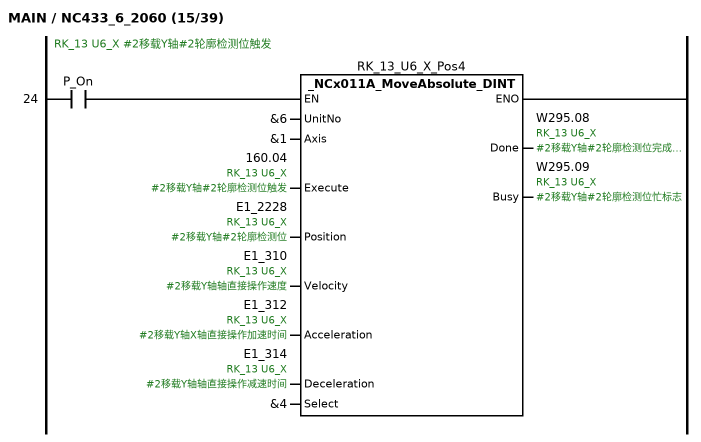
; [picture p240: MAIN / NC433_6_2060, rungs 24-24]
; rung 24: RK_13 U6_X #2移载Y轴#2轮廓检测位触发
LD P_On
CALL RK_13_U6_X_Pos4 : _NCx011A_MoveAbsolute_DINT (UnitNo := &6, Axis := &1, Execute := 160.04, Position := E1_2228, Velocity := E1_310, Acceleration := E1_312, Deceleration := E1_314, Select := &4, Done => W295.08, Busy => W295.09)  ; RK_13 U6_X #2移载Y轴#2轮廓检测位触发, RK_13 U6_X #2移载Y轴#2轮廓检测位, RK_13 U6_X #2移载Y轴轴直接操作速度, RK_13 U6_X #2移载Y轴X轴直接操作加速时间, RK_13 U6_X #2移载Y轴轴直接操作减速时间, RK_13 U6_X #2移载Y轴#2轮廓检测位完成标志, RK_13 U6_X #2移载Y轴#2轮廓检测位忙标志

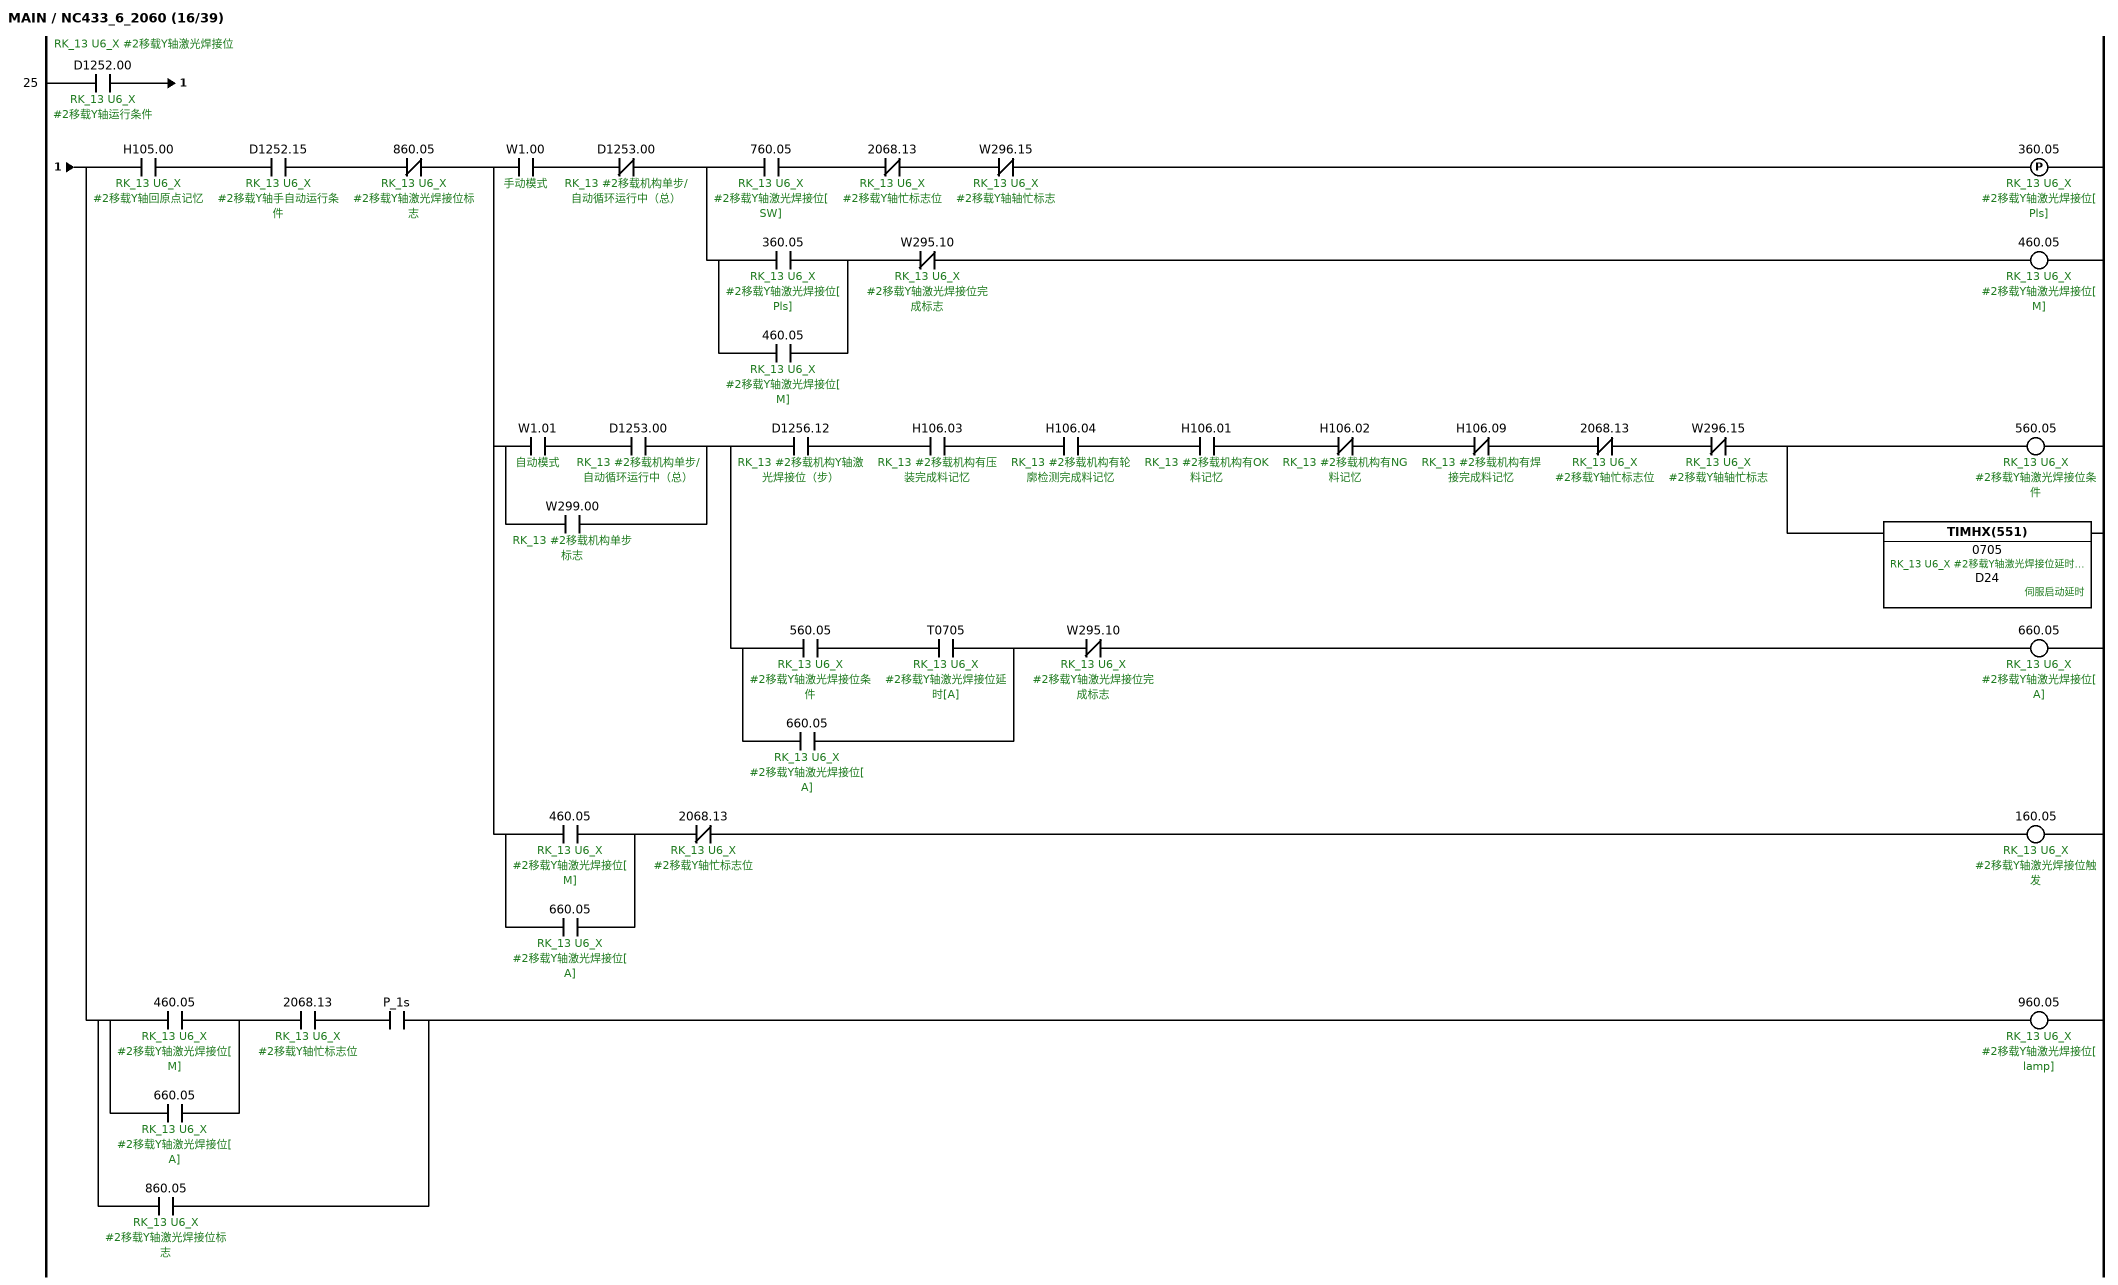
; rung 25: RK_13 U6_X #2移载Y轴激光焊接位
LD D1252.00  ; RK_13 U6_X #2移载Y轴运行条件
OUT TR0
AND H105.00  ; RK_13 U6_X #2移载Y轴回原点记忆
AND D1252.15  ; RK_13 U6_X #2移载Y轴手自动运行条件
ANDNOT 860.05  ; RK_13 U6_X #2移载Y轴激光焊接位标志
OUT TR1
AND W1.00  ; 手动模式
ANDNOT D1253.00  ; RK_13 #2移载机构单步/自动循环运行中（总）
OUT TR2
AND 760.05  ; RK_13 U6_X #2移载Y轴激光焊接位[SW]
ANDNOT 2068.13  ; RK_13 U6_X #2移载Y轴忙标志位
ANDNOT W296.15  ; RK_13 U6_X #2移载Y轴轴忙标志
DIFU(013) 360.05  ; RK_13 U6_X #2移载Y轴激光焊接位[Pls]
LD TR2
LD 360.05  ; RK_13 U6_X #2移载Y轴激光焊接位[Pls]
OR 460.05  ; RK_13 U6_X #2移载Y轴激光焊接位[M]
ANDLD
ANDNOT W295.10  ; RK_13 U6_X #2移载Y轴激光焊接位完成标志
OUT 460.05  ; RK_13 U6_X #2移载Y轴激光焊接位[M]
LD TR1
LD W1.01  ; 自动模式
AND D1253.00  ; RK_13 #2移载机构单步/自动循环运行中（总）
OR W299.00  ; RK_13 #2移载机构单步标志
ANDLD
OUT TR2
AND D1256.12  ; RK_13 #2移载机构Y轴激光焊接位（步）
AND H106.03  ; RK_13 #2移载机构有压装完成料记忆
AND H106.04  ; RK_13 #2移载机构有轮廓检测完成料记忆
AND H106.01  ; RK_13 #2移载机构有OK料记忆
ANDNOT H106.02  ; RK_13 #2移载机构有NG料记忆
ANDNOT H106.09  ; RK_13 #2移载机构有焊接完成料记忆
ANDNOT 2068.13  ; RK_13 U6_X #2移载Y轴忙标志位
ANDNOT W296.15  ; RK_13 U6_X #2移载Y轴轴忙标志
OUT 560.05  ; RK_13 U6_X #2移载Y轴激光焊接位条件
TIMHX(551) 0705 D24  ; 伺服启动延时, RK_13 U6_X #2移载Y轴激光焊接位延时[A]
LD TR2
LD 560.05  ; RK_13 U6_X #2移载Y轴激光焊接位条件
AND T0705  ; RK_13 U6_X #2移载Y轴激光焊接位延时[A]
OR 660.05  ; RK_13 U6_X #2移载Y轴激光焊接位[A]
ANDLD
ANDNOT W295.10  ; RK_13 U6_X #2移载Y轴激光焊接位完成标志
OUT 660.05  ; RK_13 U6_X #2移载Y轴激光焊接位[A]
LD TR1
LD 460.05  ; RK_13 U6_X #2移载Y轴激光焊接位[M]
OR 660.05  ; RK_13 U6_X #2移载Y轴激光焊接位[A]
ANDLD
ANDNOT 2068.13  ; RK_13 U6_X #2移载Y轴忙标志位
OUT 160.05  ; RK_13 U6_X #2移载Y轴激光焊接位触发
LD TR0
LD 460.05  ; RK_13 U6_X #2移载Y轴激光焊接位[M]
OR 660.05  ; RK_13 U6_X #2移载Y轴激光焊接位[A]
AND 2068.13  ; RK_13 U6_X #2移载Y轴忙标志位
AND P_1s
OR 860.05  ; RK_13 U6_X #2移载Y轴激光焊接位标志
ANDLD
OUT 960.05  ; RK_13 U6_X #2移载Y轴激光焊接位[lamp]

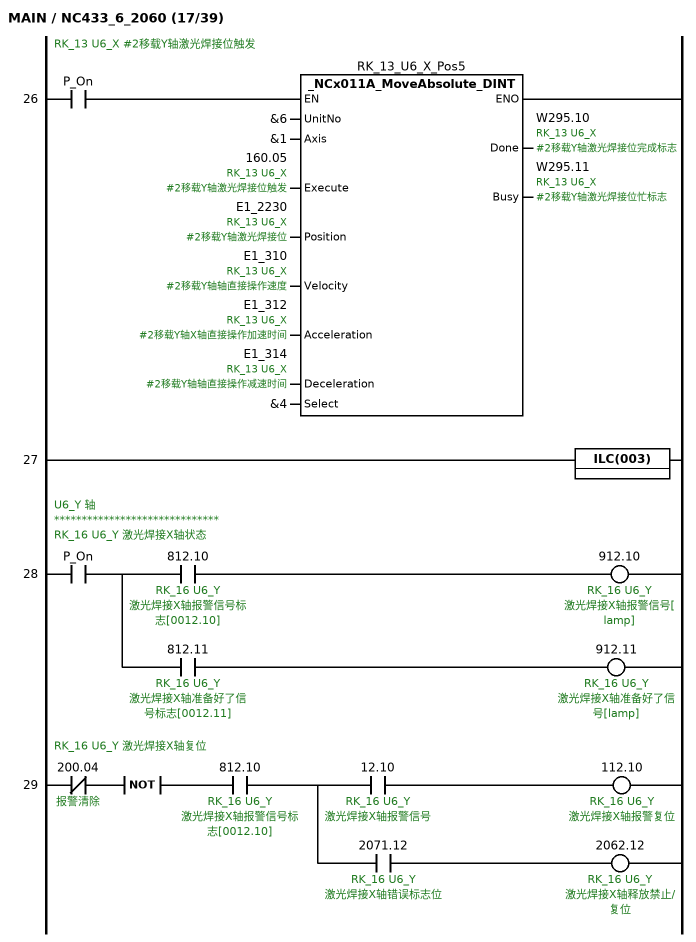
; rung 26: RK_13 U6_X #2移载Y轴激光焊接位触发
LD P_On
CALL RK_13_U6_X_Pos5 : _NCx011A_MoveAbsolute_DINT (UnitNo := &6, Axis := &1, Execute := 160.05, Position := E1_2230, Velocity := E1_310, Acceleration := E1_312, Deceleration := E1_314, Select := &4, Done => W295.10, Busy => W295.11)  ; RK_13 U6_X #2移载Y轴激光焊接位触发, RK_13 U6_X #2移载Y轴激光焊接位, RK_13 U6_X #2移载Y轴轴直接操作速度, RK_13 U6_X #2移载Y轴X轴直接操作加速时间, RK_13 U6_X #2移载Y轴轴直接操作减速时间, RK_13 U6_X #2移载Y轴激光焊接位完成标志, RK_13 U6_X #2移载Y轴激光焊接位忙标志
; rung 27
ILC(003)
; rung 28: U6_Y 轴 / ****************************** / RK_16 U6_Y 激光焊接X轴状态
LD P_On
OUT TR0
AND 812.10  ; RK_16 U6_Y 激光焊接X轴报警信号标志[0012.10]
OUT 912.10  ; RK_16 U6_Y 激光焊接X轴报警信号[lamp]
LD TR0
AND 812.11  ; RK_16 U6_Y 激光焊接X轴准备好了信号标志[0012.11]
OUT 912.11  ; RK_16 U6_Y 激光焊接X轴准备好了信号[lamp]
; rung 29: RK_16 U6_Y 激光焊接X轴复位
LDNOT 200.04  ; 报警清除
NOT(520)
AND 812.10  ; RK_16 U6_Y 激光焊接X轴报警信号标志[0012.10]
OUT TR0
AND 12.10  ; RK_16 U6_Y 激光焊接X轴报警信号
OUT 112.10  ; RK_16 U6_Y 激光焊接X轴报警复位
LD TR0
AND 2071.12  ; RK_16 U6_Y 激光焊接X轴错误标志位
OUT 2062.12  ; RK_16 U6_Y 激光焊接X轴释放禁止/复位

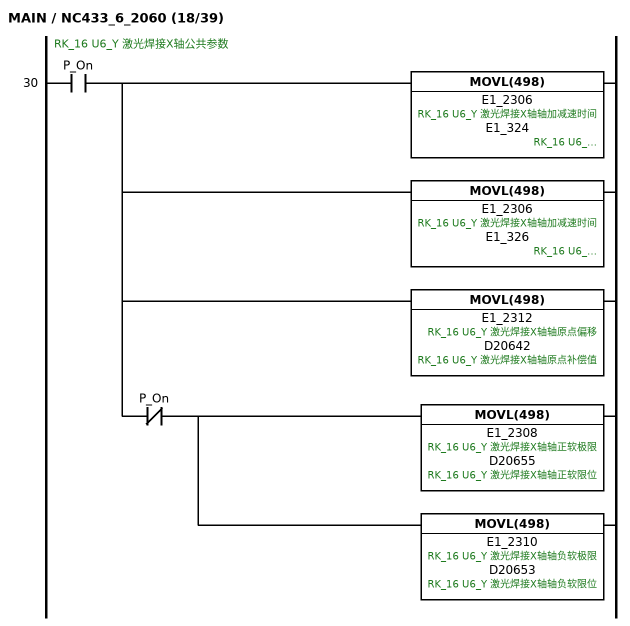
; rung 30: RK_16 U6_Y 激光焊接X轴公共参数
LD P_On
MOVL(498) E1_2306 E1_324  ; RK_16 U6_Y 激光焊接X轴轴加减速时间, RK_16 U6_Y 激光焊接X轴轴直接操作加速时间
MOVL(498) E1_2306 E1_326  ; RK_16 U6_Y 激光焊接X轴轴加减速时间, RK_16 U6_Y 激光焊接X轴轴直接操作减速时间
MOVL(498) E1_2312 D20642  ; RK_16 U6_Y 激光焊接X轴轴原点偏移, RK_16 U6_Y 激光焊接X轴轴原点补偿值
ANDNOT P_On
MOVL(498) E1_2308 D20655  ; RK_16 U6_Y 激光焊接X轴轴正软极限, RK_16 U6_Y 激光焊接X轴轴正软限位
MOVL(498) E1_2310 D20653  ; RK_16 U6_Y 激光焊接X轴轴负软极限, RK_16 U6_Y 激光焊接X轴轴负软限位

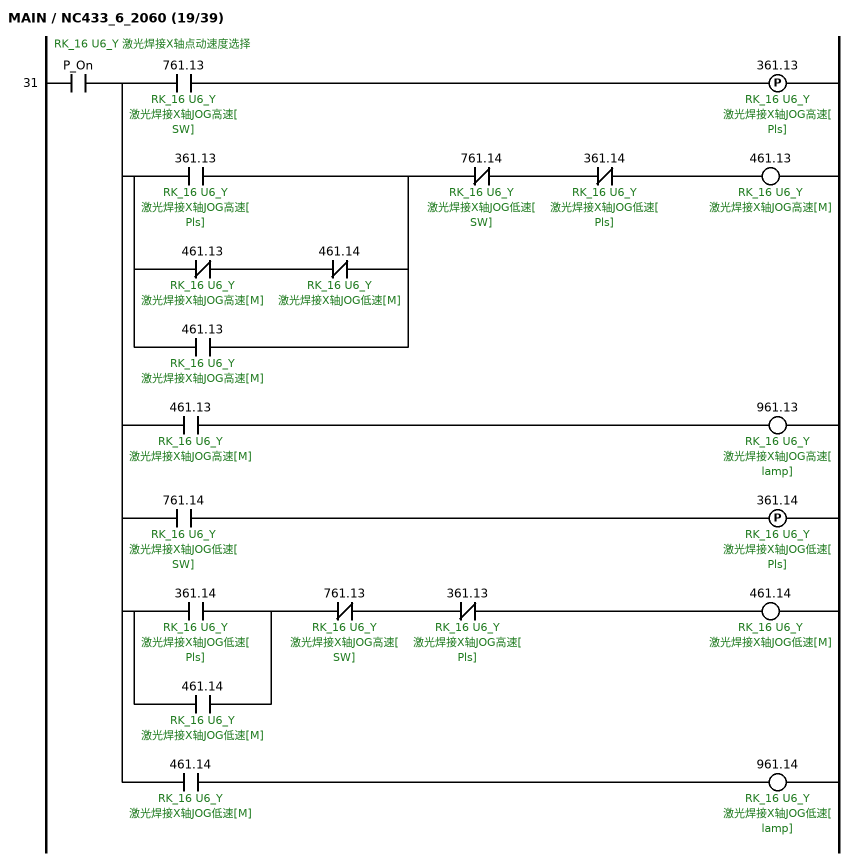
; rung 31: RK_16 U6_Y 激光焊接X轴点动速度选择
LD P_On
OUT TR0
AND 761.13  ; RK_16 U6_Y 激光焊接X轴JOG高速[SW]
DIFU(013) 361.13  ; RK_16 U6_Y 激光焊接X轴JOG高速[Pls]
LD TR0
LD 361.13  ; RK_16 U6_Y 激光焊接X轴JOG高速[Pls]
LDNOT 461.13  ; RK_16 U6_Y 激光焊接X轴JOG高速[M]
ANDNOT 461.14  ; RK_16 U6_Y 激光焊接X轴JOG低速[M]
ORLD
OR 461.13  ; RK_16 U6_Y 激光焊接X轴JOG高速[M]
ANDLD
ANDNOT 761.14  ; RK_16 U6_Y 激光焊接X轴JOG低速[SW]
ANDNOT 361.14  ; RK_16 U6_Y 激光焊接X轴JOG低速[Pls]
OUT 461.13  ; RK_16 U6_Y 激光焊接X轴JOG高速[M]
LD TR0
AND 461.13  ; RK_16 U6_Y 激光焊接X轴JOG高速[M]
OUT 961.13  ; RK_16 U6_Y 激光焊接X轴JOG高速[lamp]
LD TR0
AND 761.14  ; RK_16 U6_Y 激光焊接X轴JOG低速[SW]
DIFU(013) 361.14  ; RK_16 U6_Y 激光焊接X轴JOG低速[Pls]
LD TR0
LD 361.14  ; RK_16 U6_Y 激光焊接X轴JOG低速[Pls]
OR 461.14  ; RK_16 U6_Y 激光焊接X轴JOG低速[M]
ANDLD
ANDNOT 761.13  ; RK_16 U6_Y 激光焊接X轴JOG高速[SW]
ANDNOT 361.13  ; RK_16 U6_Y 激光焊接X轴JOG高速[Pls]
OUT 461.14  ; RK_16 U6_Y 激光焊接X轴JOG低速[M]
LD TR0
AND 461.14  ; RK_16 U6_Y 激光焊接X轴JOG低速[M]
OUT 961.14  ; RK_16 U6_Y 激光焊接X轴JOG低速[lamp]

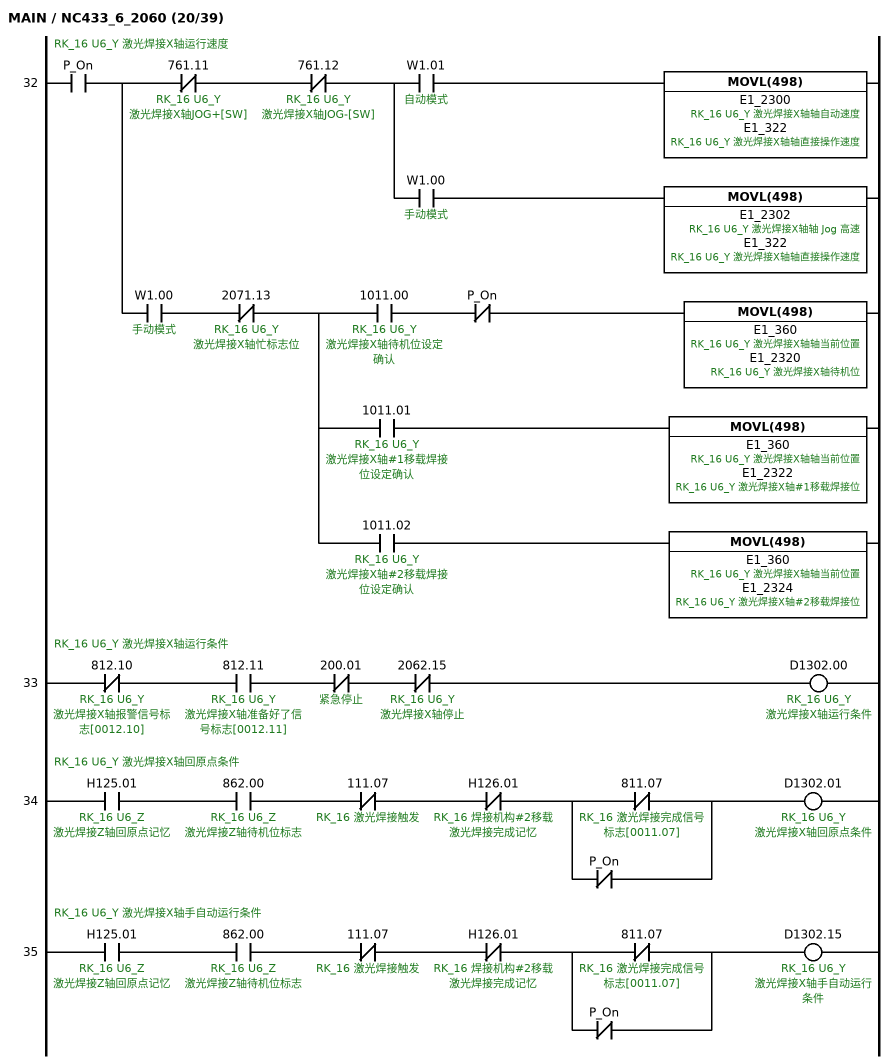
; rung 32: RK_16 U6_Y 激光焊接X轴运行速度
LD P_On
OUT TR0
ANDNOT 761.11  ; RK_16 U6_Y 激光焊接X轴JOG+[SW]
ANDNOT 761.12  ; RK_16 U6_Y 激光焊接X轴JOG-[SW]
OUT TR1
AND W1.01  ; 自动模式
MOVL(498) E1_2300 E1_322  ; RK_16 U6_Y 激光焊接X轴轴自动速度, RK_16 U6_Y 激光焊接X轴轴直接操作速度
LD TR1
AND W1.00  ; 手动模式
MOVL(498) E1_2302 E1_322  ; RK_16 U6_Y 激光焊接X轴轴 Jog 高速, RK_16 U6_Y 激光焊接X轴轴直接操作速度
LD TR0
AND W1.00  ; 手动模式
ANDNOT 2071.13  ; RK_16 U6_Y 激光焊接X轴忙标志位
OUT TR0
AND 1011.00  ; RK_16 U6_Y 激光焊接X轴待机位设定确认
ANDNOT P_On
MOVL(498) E1_360 E1_2320  ; RK_16 U6_Y 激光焊接X轴轴当前位置, RK_16 U6_Y 激光焊接X轴待机位
LD TR0
AND 1011.01  ; RK_16 U6_Y 激光焊接X轴#1移载焊接位设定确认
MOVL(498) E1_360 E1_2322  ; RK_16 U6_Y 激光焊接X轴轴当前位置, RK_16 U6_Y 激光焊接X轴#1移载焊接位
LD TR0
AND 1011.02  ; RK_16 U6_Y 激光焊接X轴#2移载焊接位设定确认
MOVL(498) E1_360 E1_2324  ; RK_16 U6_Y 激光焊接X轴轴当前位置, RK_16 U6_Y 激光焊接X轴#2移载焊接位
; rung 33: RK_16 U6_Y 激光焊接X轴运行条件
LDNOT 812.10  ; RK_16 U6_Y 激光焊接X轴报警信号标志[0012.10]
AND 812.11  ; RK_16 U6_Y 激光焊接X轴准备好了信号标志[0012.11]
ANDNOT 200.01  ; 紧急停止
ANDNOT 2062.15  ; RK_16 U6_Y 激光焊接X轴停止
OUT D1302.00  ; RK_16 U6_Y 激光焊接X轴运行条件
; rung 34: RK_16 U6_Y 激光焊接X轴回原点条件
LD H125.01  ; RK_16 U6_Z 激光焊接Z轴回原点记忆
AND 862.00  ; RK_16 U6_Z 激光焊接Z轴待机位标志
ANDNOT 111.07  ; RK_16 激光焊接触发
ANDNOT H126.01  ; RK_16 焊接机构#2移载激光焊接完成记忆
LDNOT 811.07  ; RK_16 激光焊接完成信号标志[0011.07]
ORNOT P_On
ANDLD
OUT D1302.01  ; RK_16 U6_Y 激光焊接X轴回原点条件
; rung 35: RK_16 U6_Y 激光焊接X轴手自动运行条件
LD H125.01  ; RK_16 U6_Z 激光焊接Z轴回原点记忆
AND 862.00  ; RK_16 U6_Z 激光焊接Z轴待机位标志
ANDNOT 111.07  ; RK_16 激光焊接触发
ANDNOT H126.01  ; RK_16 焊接机构#2移载激光焊接完成记忆
LDNOT 811.07  ; RK_16 激光焊接完成信号标志[0011.07]
ORNOT P_On
ANDLD
OUT D1302.15  ; RK_16 U6_Y 激光焊接X轴手自动运行条件

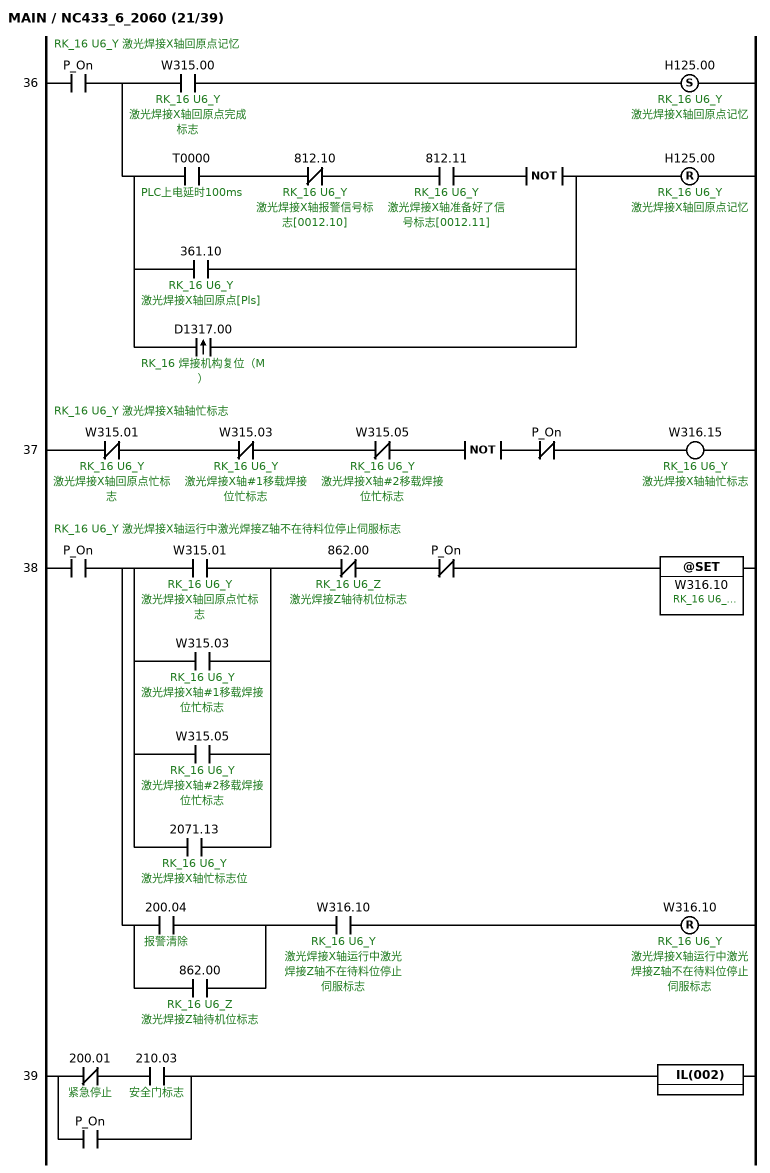
; rung 36: RK_16 U6_Y 激光焊接X轴回原点记忆
LD P_On
OUT TR0
AND W315.00  ; RK_16 U6_Y 激光焊接X轴回原点完成标志
SET H125.00  ; RK_16 U6_Y 激光焊接X轴回原点记忆
LD TR0
LD T0000  ; PLC上电延时100ms
ANDNOT 812.10  ; RK_16 U6_Y 激光焊接X轴报警信号标志[0012.10]
AND 812.11  ; RK_16 U6_Y 激光焊接X轴准备好了信号标志[0012.11]
NOT(520)
OR 361.10  ; RK_16 U6_Y 激光焊接X轴回原点[Pls]
@OR D1317.00  ; RK_16 焊接机构复位（M）
ANDLD
RSET H125.00  ; RK_16 U6_Y 激光焊接X轴回原点记忆
; rung 37: RK_16 U6_Y 激光焊接X轴轴忙标志
LDNOT W315.01  ; RK_16 U6_Y 激光焊接X轴回原点忙标志
ANDNOT W315.03  ; RK_16 U6_Y 激光焊接X轴#1移载焊接位忙标志
ANDNOT W315.05  ; RK_16 U6_Y 激光焊接X轴#2移载焊接位忙标志
NOT(520)
ANDNOT P_On
OUT W316.15  ; RK_16 U6_Y 激光焊接X轴轴忙标志
; rung 38: RK_16 U6_Y 激光焊接X轴运行中激光焊接Z轴不在待料位停止伺服标志
LD P_On
OUT TR0
LD W315.01  ; RK_16 U6_Y 激光焊接X轴回原点忙标志
OR W315.03  ; RK_16 U6_Y 激光焊接X轴#1移载焊接位忙标志
OR W315.05  ; RK_16 U6_Y 激光焊接X轴#2移载焊接位忙标志
OR 2071.13  ; RK_16 U6_Y 激光焊接X轴忙标志位
ANDLD
ANDNOT 862.00  ; RK_16 U6_Z 激光焊接Z轴待机位标志
ANDNOT P_On
@SET W316.10  ; RK_16 U6_Y 激光焊接X轴运行中激光焊接Z轴不在待料位停止伺服标志  // 增加相应报警信息
LD TR0
LD 200.04  ; 报警清除
OR 862.00  ; RK_16 U6_Z 激光焊接Z轴待机位标志
ANDLD
AND W316.10  ; RK_16 U6_Y 激光焊接X轴运行中激光焊接Z轴不在待料位停止伺服标志
RSET W316.10  ; RK_16 U6_Y 激光焊接X轴运行中激光焊接Z轴不在待料位停止伺服标志
; rung 39
LDNOT 200.01  ; 紧急停止
AND 210.03  ; 安全门标志
OR P_On
IL(002)

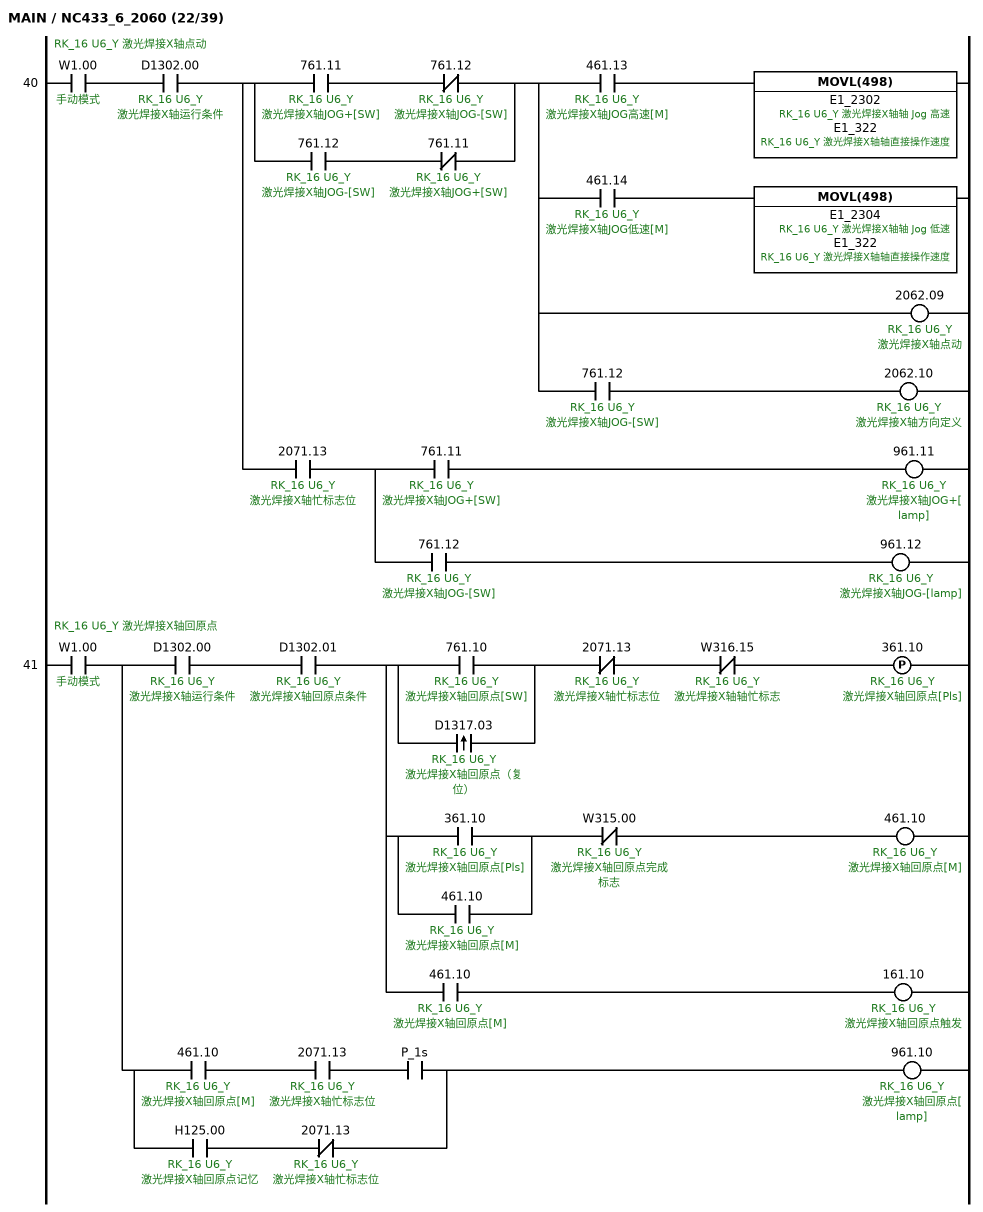
; rung 40: RK_16 U6_Y 激光焊接X轴点动
LD W1.00  ; 手动模式
AND D1302.00  ; RK_16 U6_Y 激光焊接X轴运行条件
OUT TR0
LD 761.11  ; RK_16 U6_Y 激光焊接X轴JOG+[SW]
ANDNOT 761.12  ; RK_16 U6_Y 激光焊接X轴JOG-[SW]
LD 761.12  ; RK_16 U6_Y 激光焊接X轴JOG-[SW]
ANDNOT 761.11  ; RK_16 U6_Y 激光焊接X轴JOG+[SW]
ORLD
ANDLD
OUT TR1
AND 461.13  ; RK_16 U6_Y 激光焊接X轴JOG高速[M]
MOVL(498) E1_2302 E1_322  ; RK_16 U6_Y 激光焊接X轴轴 Jog 高速, RK_16 U6_Y 激光焊接X轴轴直接操作速度
LD TR1
AND 461.14  ; RK_16 U6_Y 激光焊接X轴JOG低速[M]
MOVL(498) E1_2304 E1_322  ; RK_16 U6_Y 激光焊接X轴轴 Jog 低速, RK_16 U6_Y 激光焊接X轴轴直接操作速度
LD TR1
OUT 2062.09  ; RK_16 U6_Y 激光焊接X轴点动
AND 761.12  ; RK_16 U6_Y 激光焊接X轴JOG-[SW]
OUT 2062.10  ; RK_16 U6_Y 激光焊接X轴方向定义
LD TR0
AND 2071.13  ; RK_16 U6_Y 激光焊接X轴忙标志位
OUT TR0
AND 761.11  ; RK_16 U6_Y 激光焊接X轴JOG+[SW]
OUT 961.11  ; RK_16 U6_Y 激光焊接X轴JOG+[lamp]
LD TR0
AND 761.12  ; RK_16 U6_Y 激光焊接X轴JOG-[SW]
OUT 961.12  ; RK_16 U6_Y 激光焊接X轴JOG-[lamp]
; rung 41: RK_16 U6_Y 激光焊接X轴回原点
LD W1.00  ; 手动模式
OUT TR0
AND D1302.00  ; RK_16 U6_Y 激光焊接X轴运行条件
AND D1302.01  ; RK_16 U6_Y 激光焊接X轴回原点条件
OUT TR1
LD 761.10  ; RK_16 U6_Y 激光焊接X轴回原点[SW]
@OR D1317.03  ; RK_16 U6_Y 激光焊接X轴回原点（复位）
ANDLD
ANDNOT 2071.13  ; RK_16 U6_Y 激光焊接X轴忙标志位
ANDNOT W316.15  ; RK_16 U6_Y 激光焊接X轴轴忙标志
DIFU(013) 361.10  ; RK_16 U6_Y 激光焊接X轴回原点[Pls]
LD TR1
LD 361.10  ; RK_16 U6_Y 激光焊接X轴回原点[Pls]
OR 461.10  ; RK_16 U6_Y 激光焊接X轴回原点[M]
ANDLD
ANDNOT W315.00  ; RK_16 U6_Y 激光焊接X轴回原点完成标志
OUT 461.10  ; RK_16 U6_Y 激光焊接X轴回原点[M]
LD TR1
AND 461.10  ; RK_16 U6_Y 激光焊接X轴回原点[M]
OUT 161.10  ; RK_16 U6_Y 激光焊接X轴回原点触发
LD TR0
LD 461.10  ; RK_16 U6_Y 激光焊接X轴回原点[M]
AND 2071.13  ; RK_16 U6_Y 激光焊接X轴忙标志位
AND P_1s
LD H125.00  ; RK_16 U6_Y 激光焊接X轴回原点记忆
ANDNOT 2071.13  ; RK_16 U6_Y 激光焊接X轴忙标志位
ORLD
ANDLD
OUT 961.10  ; RK_16 U6_Y 激光焊接X轴回原点[lamp]

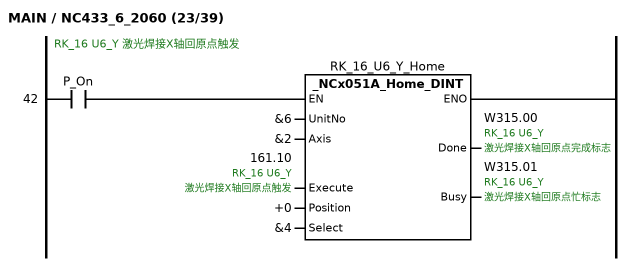
; rung 42: RK_16 U6_Y 激光焊接X轴回原点触发
LD P_On
CALL RK_16_U6_Y_Home : _NCx051A_Home_DINT (UnitNo := &6, Axis := &2, Execute := 161.10, Position := +0, Select := &4, Done => W315.00, Busy => W315.01)  ; RK_16 U6_Y 激光焊接X轴回原点触发, RK_16 U6_Y 激光焊接X轴回原点完成标志, RK_16 U6_Y 激光焊接X轴回原点忙标志

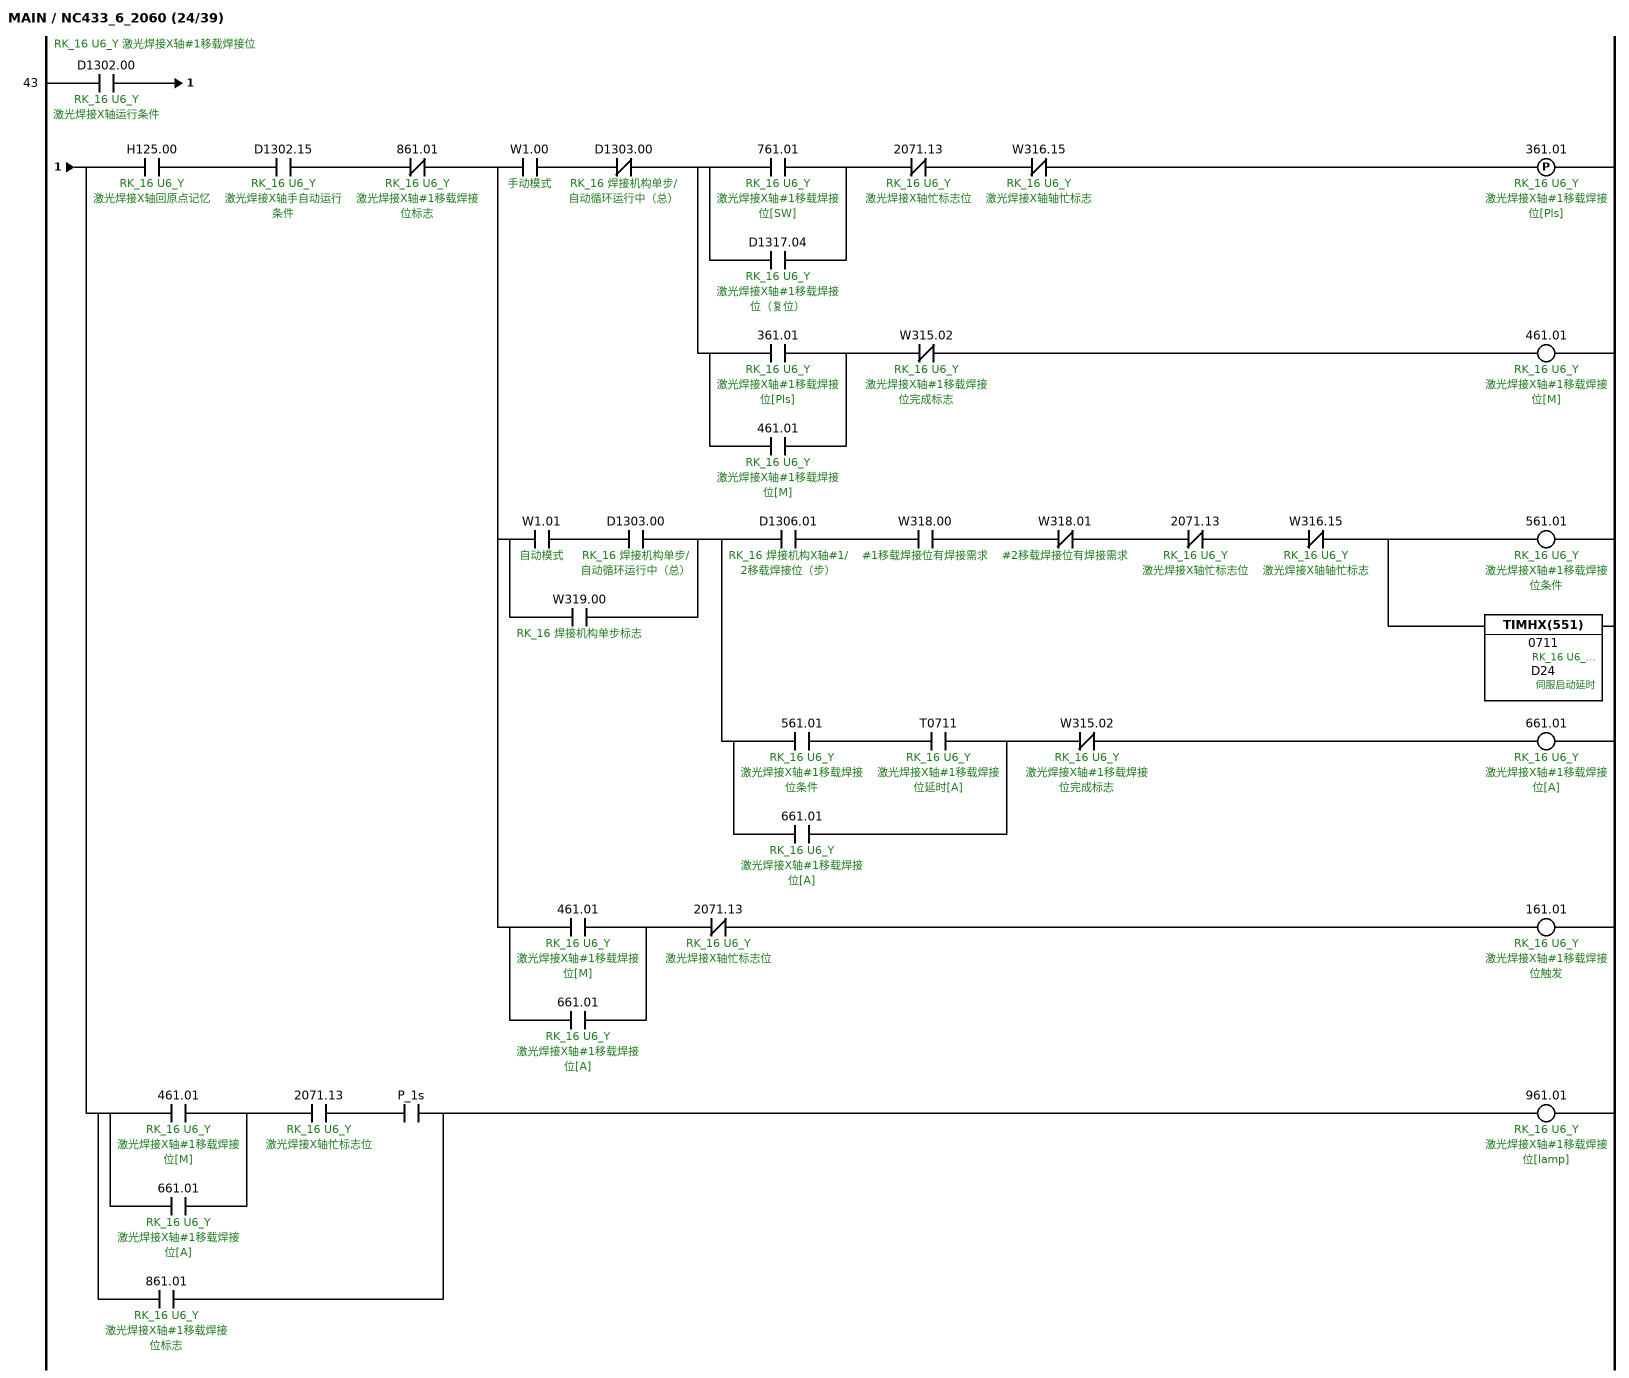
; rung 43: RK_16 U6_Y 激光焊接X轴#1移载焊接位
LD D1302.00  ; RK_16 U6_Y 激光焊接X轴运行条件
OUT TR0
AND H125.00  ; RK_16 U6_Y 激光焊接X轴回原点记忆
AND D1302.15  ; RK_16 U6_Y 激光焊接X轴手自动运行条件
ANDNOT 861.01  ; RK_16 U6_Y 激光焊接X轴#1移载焊接位标志
OUT TR1
AND W1.00  ; 手动模式
ANDNOT D1303.00  ; RK_16 焊接机构单步/自动循环运行中（总）
OUT TR2
LD 761.01  ; RK_16 U6_Y 激光焊接X轴#1移载焊接位[SW]
OR D1317.04  ; RK_16 U6_Y 激光焊接X轴#1移载焊接位（复位）
ANDLD
ANDNOT 2071.13  ; RK_16 U6_Y 激光焊接X轴忙标志位
ANDNOT W316.15  ; RK_16 U6_Y 激光焊接X轴轴忙标志
DIFU(013) 361.01  ; RK_16 U6_Y 激光焊接X轴#1移载焊接位[Pls]
LD TR2
LD 361.01  ; RK_16 U6_Y 激光焊接X轴#1移载焊接位[Pls]
OR 461.01  ; RK_16 U6_Y 激光焊接X轴#1移载焊接位[M]
ANDLD
ANDNOT W315.02  ; RK_16 U6_Y 激光焊接X轴#1移载焊接位完成标志
OUT 461.01  ; RK_16 U6_Y 激光焊接X轴#1移载焊接位[M]
LD TR1
LD W1.01  ; 自动模式
AND D1303.00  ; RK_16 焊接机构单步/自动循环运行中（总）
OR W319.00  ; RK_16 焊接机构单步标志
ANDLD
OUT TR2
AND D1306.01  ; RK_16 焊接机构X轴#1/2移载焊接位（步）
AND W318.00  ; #1移载焊接位有焊接需求
ANDNOT W318.01  ; #2移载焊接位有焊接需求
ANDNOT 2071.13  ; RK_16 U6_Y 激光焊接X轴忙标志位
ANDNOT W316.15  ; RK_16 U6_Y 激光焊接X轴轴忙标志
OUT 561.01  ; RK_16 U6_Y 激光焊接X轴#1移载焊接位条件
TIMHX(551) 0711 D24  ; 伺服启动延时, RK_16 U6_Y 激光焊接X轴#1移载焊接位延时[A]
LD TR2
LD 561.01  ; RK_16 U6_Y 激光焊接X轴#1移载焊接位条件
AND T0711  ; RK_16 U6_Y 激光焊接X轴#1移载焊接位延时[A]
OR 661.01  ; RK_16 U6_Y 激光焊接X轴#1移载焊接位[A]
ANDLD
ANDNOT W315.02  ; RK_16 U6_Y 激光焊接X轴#1移载焊接位完成标志
OUT 661.01  ; RK_16 U6_Y 激光焊接X轴#1移载焊接位[A]
LD TR1
LD 461.01  ; RK_16 U6_Y 激光焊接X轴#1移载焊接位[M]
OR 661.01  ; RK_16 U6_Y 激光焊接X轴#1移载焊接位[A]
ANDLD
ANDNOT 2071.13  ; RK_16 U6_Y 激光焊接X轴忙标志位
OUT 161.01  ; RK_16 U6_Y 激光焊接X轴#1移载焊接位触发
LD TR0
LD 461.01  ; RK_16 U6_Y 激光焊接X轴#1移载焊接位[M]
OR 661.01  ; RK_16 U6_Y 激光焊接X轴#1移载焊接位[A]
AND 2071.13  ; RK_16 U6_Y 激光焊接X轴忙标志位
AND P_1s
OR 861.01  ; RK_16 U6_Y 激光焊接X轴#1移载焊接位标志
ANDLD
OUT 961.01  ; RK_16 U6_Y 激光焊接X轴#1移载焊接位[lamp]

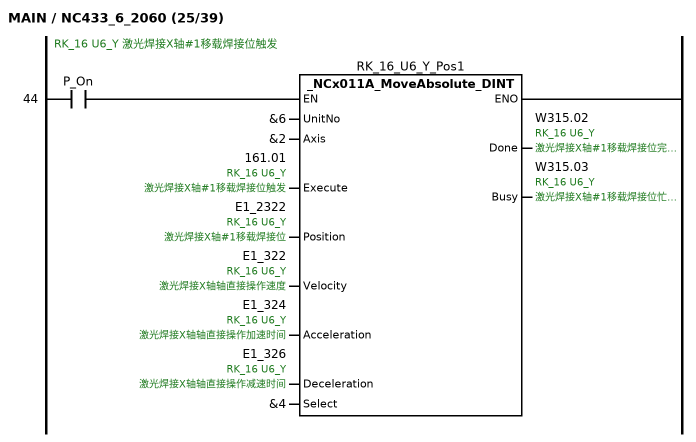
; rung 44: RK_16 U6_Y 激光焊接X轴#1移载焊接位触发
LD P_On
CALL RK_16_U6_Y_Pos1 : _NCx011A_MoveAbsolute_DINT (UnitNo := &6, Axis := &2, Execute := 161.01, Position := E1_2322, Velocity := E1_322, Acceleration := E1_324, Deceleration := E1_326, Select := &4, Done => W315.02, Busy => W315.03)  ; RK_16 U6_Y 激光焊接X轴#1移载焊接位触发, RK_16 U6_Y 激光焊接X轴#1移载焊接位, RK_16 U6_Y 激光焊接X轴轴直接操作速度, RK_16 U6_Y 激光焊接X轴轴直接操作加速时间, RK_16 U6_Y 激光焊接X轴轴直接操作减速时间, RK_16 U6_Y 激光焊接X轴#1移载焊接位完成标志, RK_16 U6_Y 激光焊接X轴#1移载焊接位忙标志

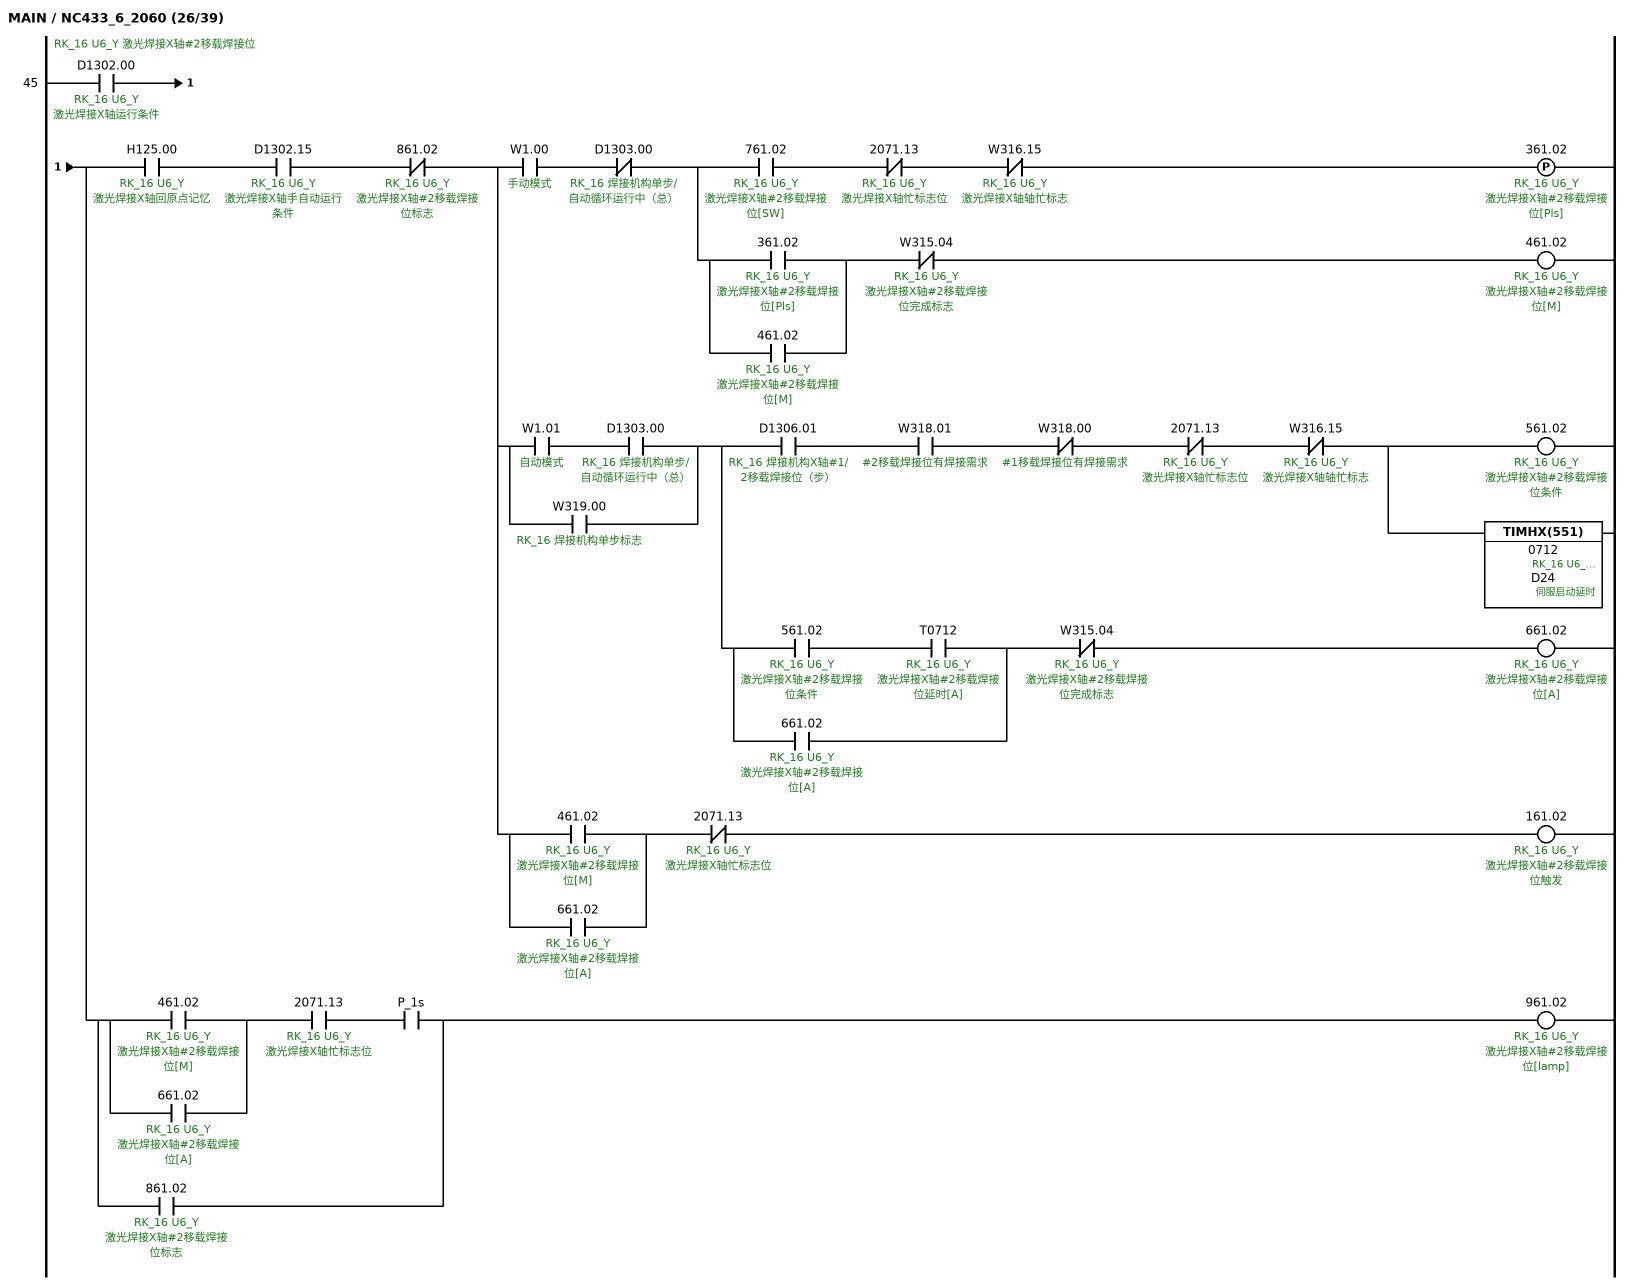
; rung 45: RK_16 U6_Y 激光焊接X轴#2移载焊接位
LD D1302.00  ; RK_16 U6_Y 激光焊接X轴运行条件
OUT TR0
AND H125.00  ; RK_16 U6_Y 激光焊接X轴回原点记忆
AND D1302.15  ; RK_16 U6_Y 激光焊接X轴手自动运行条件
ANDNOT 861.02  ; RK_16 U6_Y 激光焊接X轴#2移载焊接位标志
OUT TR1
AND W1.00  ; 手动模式
ANDNOT D1303.00  ; RK_16 焊接机构单步/自动循环运行中（总）
OUT TR2
AND 761.02  ; RK_16 U6_Y 激光焊接X轴#2移载焊接位[SW]
ANDNOT 2071.13  ; RK_16 U6_Y 激光焊接X轴忙标志位
ANDNOT W316.15  ; RK_16 U6_Y 激光焊接X轴轴忙标志
DIFU(013) 361.02  ; RK_16 U6_Y 激光焊接X轴#2移载焊接位[Pls]
LD TR2
LD 361.02  ; RK_16 U6_Y 激光焊接X轴#2移载焊接位[Pls]
OR 461.02  ; RK_16 U6_Y 激光焊接X轴#2移载焊接位[M]
ANDLD
ANDNOT W315.04  ; RK_16 U6_Y 激光焊接X轴#2移载焊接位完成标志
OUT 461.02  ; RK_16 U6_Y 激光焊接X轴#2移载焊接位[M]
LD TR1
LD W1.01  ; 自动模式
AND D1303.00  ; RK_16 焊接机构单步/自动循环运行中（总）
OR W319.00  ; RK_16 焊接机构单步标志
ANDLD
OUT TR2
AND D1306.01  ; RK_16 焊接机构X轴#1/2移载焊接位（步）
AND W318.01  ; #2移载焊接位有焊接需求
ANDNOT W318.00  ; #1移载焊接位有焊接需求
ANDNOT 2071.13  ; RK_16 U6_Y 激光焊接X轴忙标志位
ANDNOT W316.15  ; RK_16 U6_Y 激光焊接X轴轴忙标志
OUT 561.02  ; RK_16 U6_Y 激光焊接X轴#2移载焊接位条件
TIMHX(551) 0712 D24  ; 伺服启动延时, RK_16 U6_Y 激光焊接X轴#2移载焊接位延时[A]
LD TR2
LD 561.02  ; RK_16 U6_Y 激光焊接X轴#2移载焊接位条件
AND T0712  ; RK_16 U6_Y 激光焊接X轴#2移载焊接位延时[A]
OR 661.02  ; RK_16 U6_Y 激光焊接X轴#2移载焊接位[A]
ANDLD
ANDNOT W315.04  ; RK_16 U6_Y 激光焊接X轴#2移载焊接位完成标志
OUT 661.02  ; RK_16 U6_Y 激光焊接X轴#2移载焊接位[A]
LD TR1
LD 461.02  ; RK_16 U6_Y 激光焊接X轴#2移载焊接位[M]
OR 661.02  ; RK_16 U6_Y 激光焊接X轴#2移载焊接位[A]
ANDLD
ANDNOT 2071.13  ; RK_16 U6_Y 激光焊接X轴忙标志位
OUT 161.02  ; RK_16 U6_Y 激光焊接X轴#2移载焊接位触发
LD TR0
LD 461.02  ; RK_16 U6_Y 激光焊接X轴#2移载焊接位[M]
OR 661.02  ; RK_16 U6_Y 激光焊接X轴#2移载焊接位[A]
AND 2071.13  ; RK_16 U6_Y 激光焊接X轴忙标志位
AND P_1s
OR 861.02  ; RK_16 U6_Y 激光焊接X轴#2移载焊接位标志
ANDLD
OUT 961.02  ; RK_16 U6_Y 激光焊接X轴#2移载焊接位[lamp]

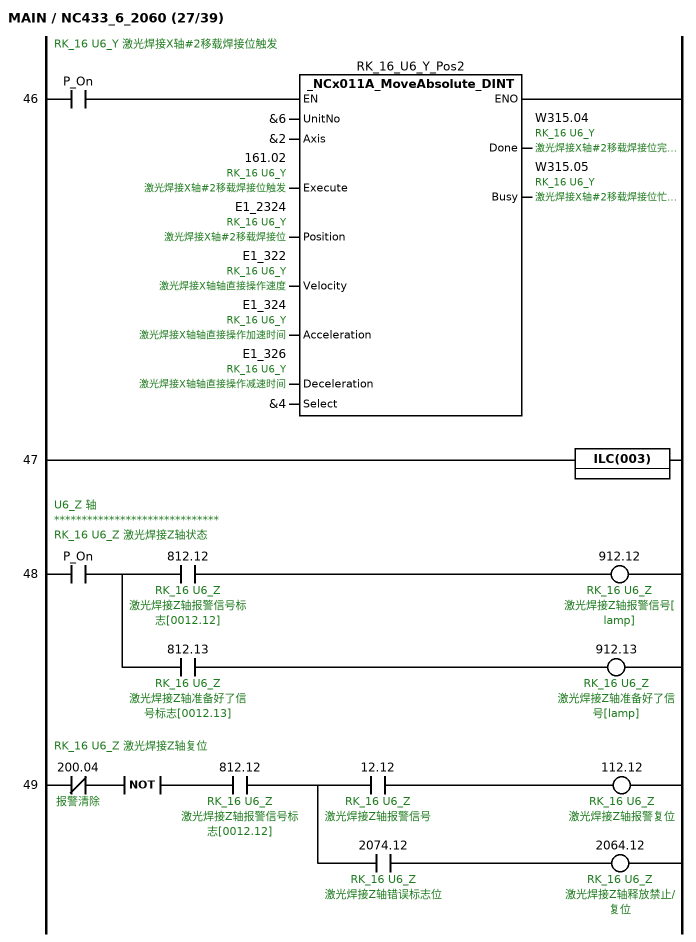
; rung 46: RK_16 U6_Y 激光焊接X轴#2移载焊接位触发
LD P_On
CALL RK_16_U6_Y_Pos2 : _NCx011A_MoveAbsolute_DINT (UnitNo := &6, Axis := &2, Execute := 161.02, Position := E1_2324, Velocity := E1_322, Acceleration := E1_324, Deceleration := E1_326, Select := &4, Done => W315.04, Busy => W315.05)  ; RK_16 U6_Y 激光焊接X轴#2移载焊接位触发, RK_16 U6_Y 激光焊接X轴#2移载焊接位, RK_16 U6_Y 激光焊接X轴轴直接操作速度, RK_16 U6_Y 激光焊接X轴轴直接操作加速时间, RK_16 U6_Y 激光焊接X轴轴直接操作减速时间, RK_16 U6_Y 激光焊接X轴#2移载焊接位完成标志, RK_16 U6_Y 激光焊接X轴#2移载焊接位忙标志
; rung 47
ILC(003)
; rung 48: U6_Z 轴 / ****************************** / RK_16 U6_Z 激光焊接Z轴状态
LD P_On
OUT TR0
AND 812.12  ; RK_16 U6_Z 激光焊接Z轴报警信号标志[0012.12]
OUT 912.12  ; RK_16 U6_Z 激光焊接Z轴报警信号[lamp]
LD TR0
AND 812.13  ; RK_16 U6_Z 激光焊接Z轴准备好了信号标志[0012.13]
OUT 912.13  ; RK_16 U6_Z 激光焊接Z轴准备好了信号[lamp]
; rung 49: RK_16 U6_Z 激光焊接Z轴复位
LDNOT 200.04  ; 报警清除
NOT(520)
AND 812.12  ; RK_16 U6_Z 激光焊接Z轴报警信号标志[0012.12]
OUT TR0
AND 12.12  ; RK_16 U6_Z 激光焊接Z轴报警信号
OUT 112.12  ; RK_16 U6_Z 激光焊接Z轴报警复位
LD TR0
AND 2074.12  ; RK_16 U6_Z 激光焊接Z轴错误标志位
OUT 2064.12  ; RK_16 U6_Z 激光焊接Z轴释放禁止/复位

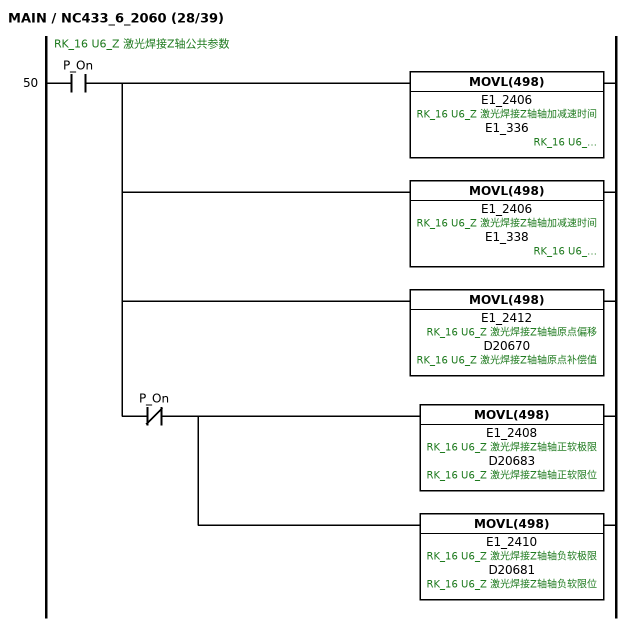
; rung 50: RK_16 U6_Z 激光焊接Z轴公共参数
LD P_On
MOVL(498) E1_2406 E1_336  ; RK_16 U6_Z 激光焊接Z轴轴加减速时间, RK_16 U6_Z 激光焊接Z轴轴直接操作加速时间
MOVL(498) E1_2406 E1_338  ; RK_16 U6_Z 激光焊接Z轴轴加减速时间, RK_16 U6_Z 激光焊接Z轴轴直接操作减速时间
MOVL(498) E1_2412 D20670  ; RK_16 U6_Z 激光焊接Z轴轴原点偏移, RK_16 U6_Z 激光焊接Z轴轴原点补偿值
ANDNOT P_On
MOVL(498) E1_2408 D20683  ; RK_16 U6_Z 激光焊接Z轴轴正软极限, RK_16 U6_Z 激光焊接Z轴轴正软限位
MOVL(498) E1_2410 D20681  ; RK_16 U6_Z 激光焊接Z轴轴负软极限, RK_16 U6_Z 激光焊接Z轴轴负软限位

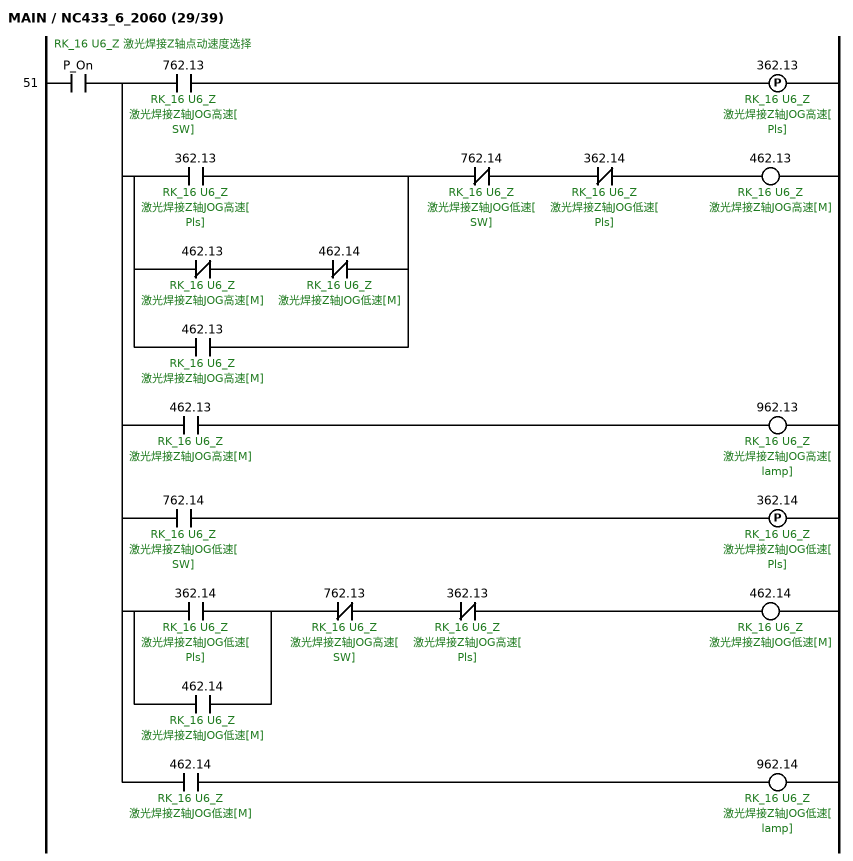
; rung 51: RK_16 U6_Z 激光焊接Z轴点动速度选择
LD P_On
OUT TR0
AND 762.13  ; RK_16 U6_Z 激光焊接Z轴JOG高速[SW]
DIFU(013) 362.13  ; RK_16 U6_Z 激光焊接Z轴JOG高速[Pls]
LD TR0
LD 362.13  ; RK_16 U6_Z 激光焊接Z轴JOG高速[Pls]
LDNOT 462.13  ; RK_16 U6_Z 激光焊接Z轴JOG高速[M]
ANDNOT 462.14  ; RK_16 U6_Z 激光焊接Z轴JOG低速[M]
ORLD
OR 462.13  ; RK_16 U6_Z 激光焊接Z轴JOG高速[M]
ANDLD
ANDNOT 762.14  ; RK_16 U6_Z 激光焊接Z轴JOG低速[SW]
ANDNOT 362.14  ; RK_16 U6_Z 激光焊接Z轴JOG低速[Pls]
OUT 462.13  ; RK_16 U6_Z 激光焊接Z轴JOG高速[M]
LD TR0
AND 462.13  ; RK_16 U6_Z 激光焊接Z轴JOG高速[M]
OUT 962.13  ; RK_16 U6_Z 激光焊接Z轴JOG高速[lamp]
LD TR0
AND 762.14  ; RK_16 U6_Z 激光焊接Z轴JOG低速[SW]
DIFU(013) 362.14  ; RK_16 U6_Z 激光焊接Z轴JOG低速[Pls]
LD TR0
LD 362.14  ; RK_16 U6_Z 激光焊接Z轴JOG低速[Pls]
OR 462.14  ; RK_16 U6_Z 激光焊接Z轴JOG低速[M]
ANDLD
ANDNOT 762.13  ; RK_16 U6_Z 激光焊接Z轴JOG高速[SW]
ANDNOT 362.13  ; RK_16 U6_Z 激光焊接Z轴JOG高速[Pls]
OUT 462.14  ; RK_16 U6_Z 激光焊接Z轴JOG低速[M]
LD TR0
AND 462.14  ; RK_16 U6_Z 激光焊接Z轴JOG低速[M]
OUT 962.14  ; RK_16 U6_Z 激光焊接Z轴JOG低速[lamp]

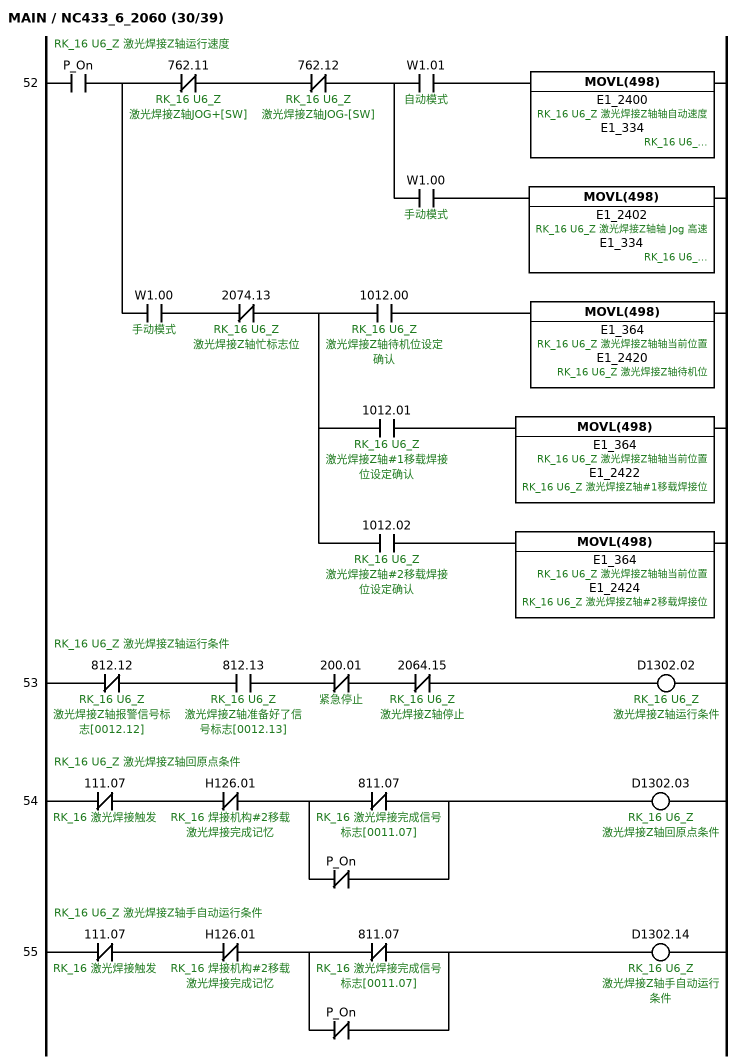
; rung 52: RK_16 U6_Z 激光焊接Z轴运行速度
LD P_On
OUT TR0
ANDNOT 762.11  ; RK_16 U6_Z 激光焊接Z轴JOG+[SW]
ANDNOT 762.12  ; RK_16 U6_Z 激光焊接Z轴JOG-[SW]
OUT TR1
AND W1.01  ; 自动模式
MOVL(498) E1_2400 E1_334  ; RK_16 U6_Z 激光焊接Z轴轴自动速度, RK_16 U6_Z 激光焊接Z轴轴直接操作速度
LD TR1
AND W1.00  ; 手动模式
MOVL(498) E1_2402 E1_334  ; RK_16 U6_Z 激光焊接Z轴轴 Jog 高速, RK_16 U6_Z 激光焊接Z轴轴直接操作速度
LD TR0
AND W1.00  ; 手动模式
ANDNOT 2074.13  ; RK_16 U6_Z 激光焊接Z轴忙标志位
OUT TR0
AND 1012.00  ; RK_16 U6_Z 激光焊接Z轴待机位设定确认
MOVL(498) E1_364 E1_2420  ; RK_16 U6_Z 激光焊接Z轴轴当前位置, RK_16 U6_Z 激光焊接Z轴待机位
LD TR0
AND 1012.01  ; RK_16 U6_Z 激光焊接Z轴#1移载焊接位设定确认
MOVL(498) E1_364 E1_2422  ; RK_16 U6_Z 激光焊接Z轴轴当前位置, RK_16 U6_Z 激光焊接Z轴#1移载焊接位
LD TR0
AND 1012.02  ; RK_16 U6_Z 激光焊接Z轴#2移载焊接位设定确认
MOVL(498) E1_364 E1_2424  ; RK_16 U6_Z 激光焊接Z轴轴当前位置, RK_16 U6_Z 激光焊接Z轴#2移载焊接位
; rung 53: RK_16 U6_Z 激光焊接Z轴运行条件
LDNOT 812.12  ; RK_16 U6_Z 激光焊接Z轴报警信号标志[0012.12]
AND 812.13  ; RK_16 U6_Z 激光焊接Z轴准备好了信号标志[0012.13]
ANDNOT 200.01  ; 紧急停止
ANDNOT 2064.15  ; RK_16 U6_Z 激光焊接Z轴停止
OUT D1302.02  ; RK_16 U6_Z 激光焊接Z轴运行条件
; rung 54: RK_16 U6_Z 激光焊接Z轴回原点条件
LDNOT 111.07  ; RK_16 激光焊接触发
ANDNOT H126.01  ; RK_16 焊接机构#2移载激光焊接完成记忆
LDNOT 811.07  ; RK_16 激光焊接完成信号标志[0011.07]
ORNOT P_On
ANDLD
OUT D1302.03  ; RK_16 U6_Z 激光焊接Z轴回原点条件
; rung 55: RK_16 U6_Z 激光焊接Z轴手自动运行条件
LDNOT 111.07  ; RK_16 激光焊接触发
ANDNOT H126.01  ; RK_16 焊接机构#2移载激光焊接完成记忆
LDNOT 811.07  ; RK_16 激光焊接完成信号标志[0011.07]
ORNOT P_On
ANDLD
OUT D1302.14  ; RK_16 U6_Z 激光焊接Z轴手自动运行条件

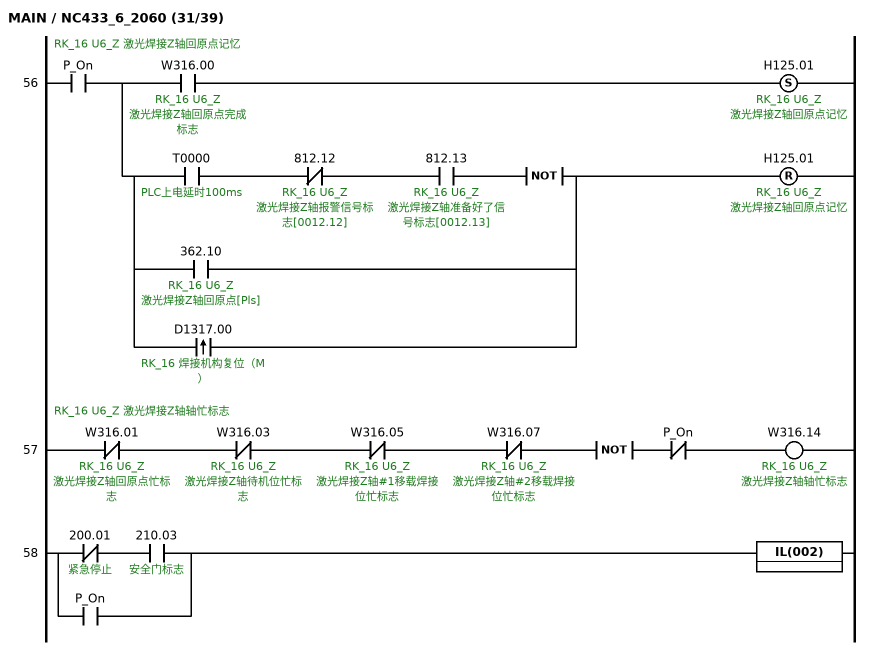
; rung 56: RK_16 U6_Z 激光焊接Z轴回原点记忆
LD P_On
OUT TR0
AND W316.00  ; RK_16 U6_Z 激光焊接Z轴回原点完成标志
SET H125.01  ; RK_16 U6_Z 激光焊接Z轴回原点记忆
LD TR0
LD T0000  ; PLC上电延时100ms
ANDNOT 812.12  ; RK_16 U6_Z 激光焊接Z轴报警信号标志[0012.12]
AND 812.13  ; RK_16 U6_Z 激光焊接Z轴准备好了信号标志[0012.13]
NOT(520)
OR 362.10  ; RK_16 U6_Z 激光焊接Z轴回原点[Pls]
@OR D1317.00  ; RK_16 焊接机构复位（M）
ANDLD
RSET H125.01  ; RK_16 U6_Z 激光焊接Z轴回原点记忆
; rung 57: RK_16 U6_Z 激光焊接Z轴轴忙标志
LDNOT W316.01  ; RK_16 U6_Z 激光焊接Z轴回原点忙标志
ANDNOT W316.03  ; RK_16 U6_Z 激光焊接Z轴待机位忙标志
ANDNOT W316.05  ; RK_16 U6_Z 激光焊接Z轴#1移载焊接位忙标志
ANDNOT W316.07  ; RK_16 U6_Z 激光焊接Z轴#2移载焊接位忙标志
NOT(520)
ANDNOT P_On
OUT W316.14  ; RK_16 U6_Z 激光焊接Z轴轴忙标志
; rung 58
LDNOT 200.01  ; 紧急停止
AND 210.03  ; 安全门标志
OR P_On
IL(002)

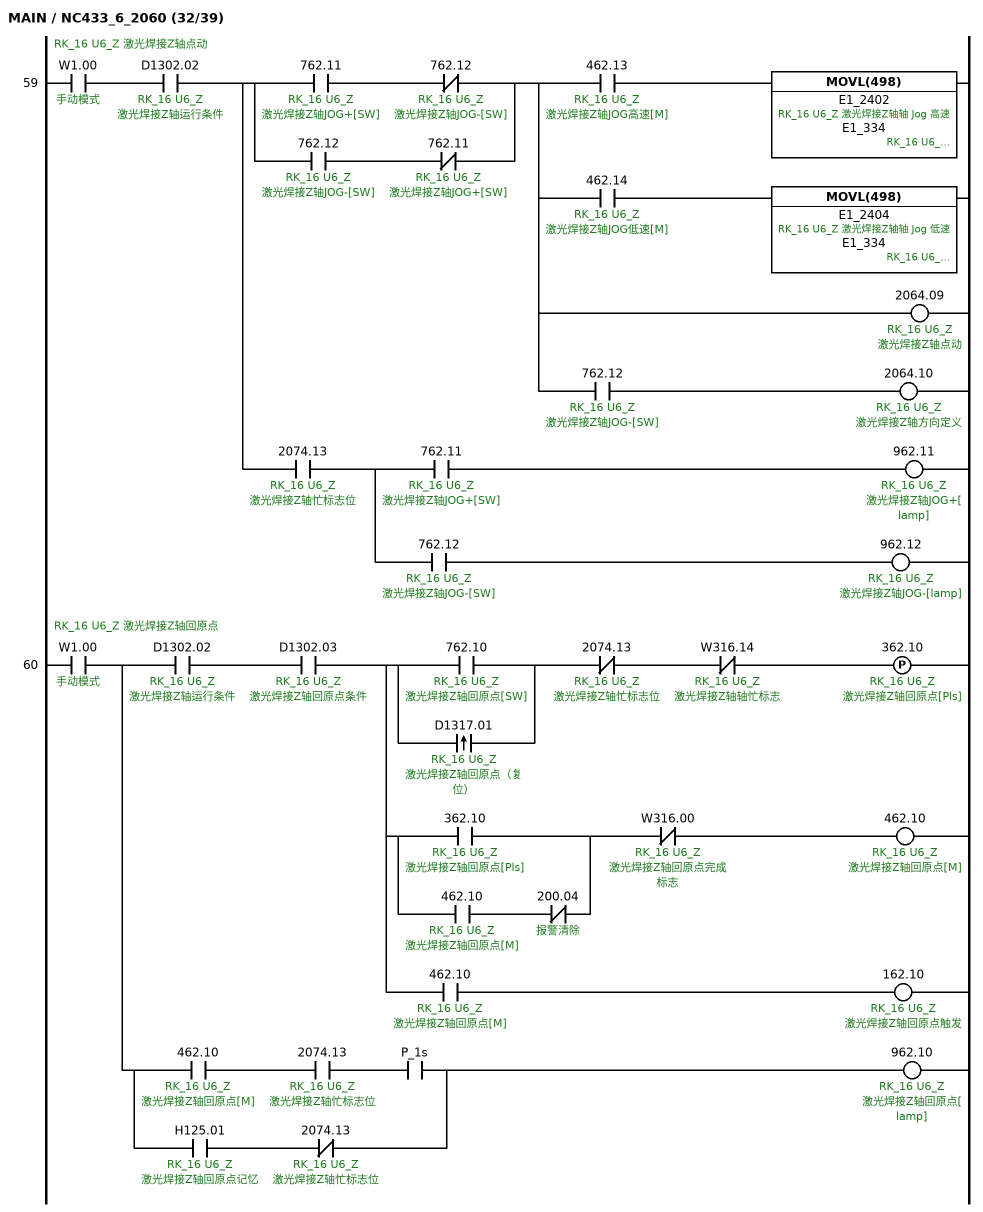
; rung 59: RK_16 U6_Z 激光焊接Z轴点动
LD W1.00  ; 手动模式
AND D1302.02  ; RK_16 U6_Z 激光焊接Z轴运行条件
OUT TR0
LD 762.11  ; RK_16 U6_Z 激光焊接Z轴JOG+[SW]
ANDNOT 762.12  ; RK_16 U6_Z 激光焊接Z轴JOG-[SW]
LD 762.12  ; RK_16 U6_Z 激光焊接Z轴JOG-[SW]
ANDNOT 762.11  ; RK_16 U6_Z 激光焊接Z轴JOG+[SW]
ORLD
ANDLD
OUT TR1
AND 462.13  ; RK_16 U6_Z 激光焊接Z轴JOG高速[M]
MOVL(498) E1_2402 E1_334  ; RK_16 U6_Z 激光焊接Z轴轴 Jog 高速, RK_16 U6_Z 激光焊接Z轴轴直接操作速度
LD TR1
AND 462.14  ; RK_16 U6_Z 激光焊接Z轴JOG低速[M]
MOVL(498) E1_2404 E1_334  ; RK_16 U6_Z 激光焊接Z轴轴 Jog 低速, RK_16 U6_Z 激光焊接Z轴轴直接操作速度
LD TR1
OUT 2064.09  ; RK_16 U6_Z 激光焊接Z轴点动
AND 762.12  ; RK_16 U6_Z 激光焊接Z轴JOG-[SW]
OUT 2064.10  ; RK_16 U6_Z 激光焊接Z轴方向定义
LD TR0
AND 2074.13  ; RK_16 U6_Z 激光焊接Z轴忙标志位
OUT TR0
AND 762.11  ; RK_16 U6_Z 激光焊接Z轴JOG+[SW]
OUT 962.11  ; RK_16 U6_Z 激光焊接Z轴JOG+[lamp]
LD TR0
AND 762.12  ; RK_16 U6_Z 激光焊接Z轴JOG-[SW]
OUT 962.12  ; RK_16 U6_Z 激光焊接Z轴JOG-[lamp]
; rung 60: RK_16 U6_Z 激光焊接Z轴回原点
LD W1.00  ; 手动模式
OUT TR0
AND D1302.02  ; RK_16 U6_Z 激光焊接Z轴运行条件
AND D1302.03  ; RK_16 U6_Z 激光焊接Z轴回原点条件
OUT TR1
LD 762.10  ; RK_16 U6_Z 激光焊接Z轴回原点[SW]
@OR D1317.01  ; RK_16 U6_Z 激光焊接Z轴回原点（复位）
ANDLD
ANDNOT 2074.13  ; RK_16 U6_Z 激光焊接Z轴忙标志位
ANDNOT W316.14  ; RK_16 U6_Z 激光焊接Z轴轴忙标志
DIFU(013) 362.10  ; RK_16 U6_Z 激光焊接Z轴回原点[Pls]
LD TR1
LD 362.10  ; RK_16 U6_Z 激光焊接Z轴回原点[Pls]
LD 462.10  ; RK_16 U6_Z 激光焊接Z轴回原点[M]
ANDNOT 200.04  ; 报警清除
ORLD
ANDLD
ANDNOT W316.00  ; RK_16 U6_Z 激光焊接Z轴回原点完成标志
OUT 462.10  ; RK_16 U6_Z 激光焊接Z轴回原点[M]
LD TR1
AND 462.10  ; RK_16 U6_Z 激光焊接Z轴回原点[M]
OUT 162.10  ; RK_16 U6_Z 激光焊接Z轴回原点触发
LD TR0
LD 462.10  ; RK_16 U6_Z 激光焊接Z轴回原点[M]
AND 2074.13  ; RK_16 U6_Z 激光焊接Z轴忙标志位
AND P_1s
LD H125.01  ; RK_16 U6_Z 激光焊接Z轴回原点记忆
ANDNOT 2074.13  ; RK_16 U6_Z 激光焊接Z轴忙标志位
ORLD
ANDLD
OUT 962.10  ; RK_16 U6_Z 激光焊接Z轴回原点[lamp]

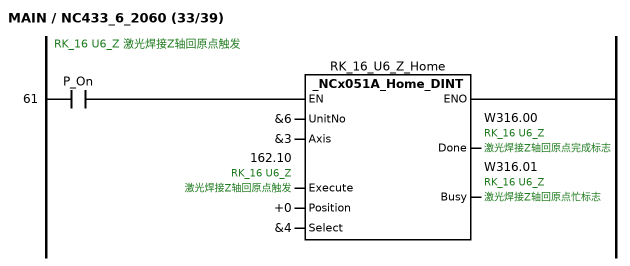
; rung 61: RK_16 U6_Z 激光焊接Z轴回原点触发
LD P_On
CALL RK_16_U6_Z_Home : _NCx051A_Home_DINT (UnitNo := &6, Axis := &3, Execute := 162.10, Position := +0, Select := &4, Done => W316.00, Busy => W316.01)  ; RK_16 U6_Z 激光焊接Z轴回原点触发, RK_16 U6_Z 激光焊接Z轴回原点完成标志, RK_16 U6_Z 激光焊接Z轴回原点忙标志

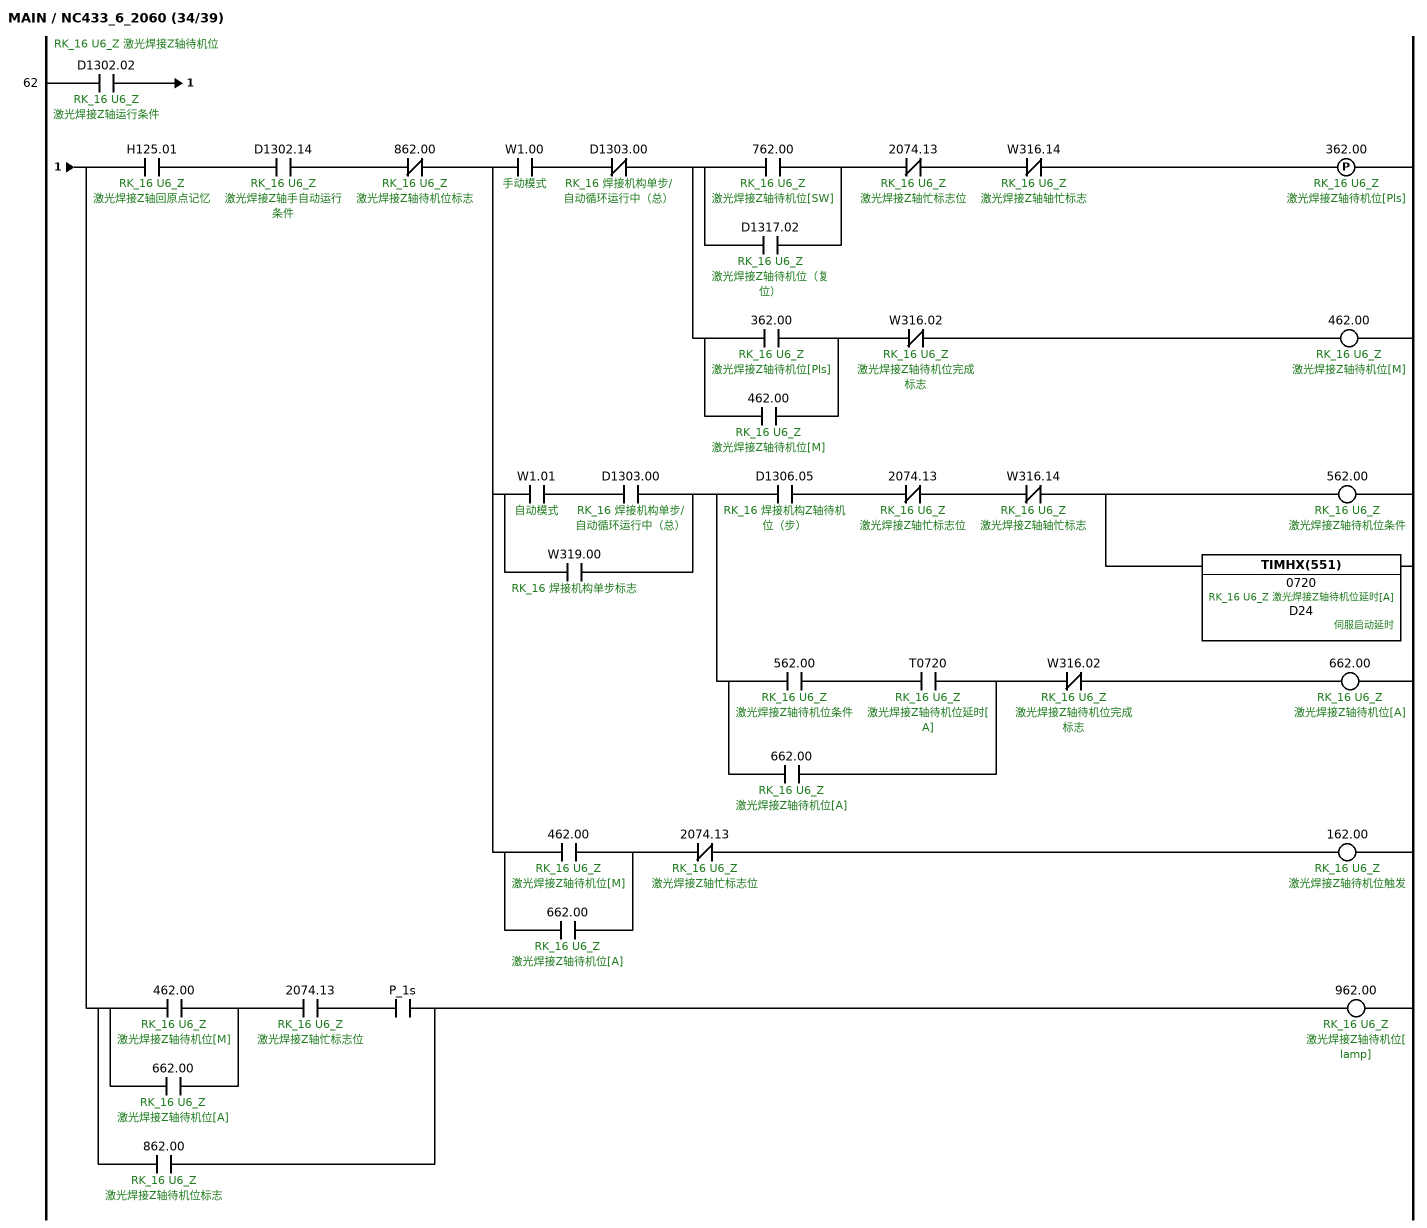
; rung 62: RK_16 U6_Z 激光焊接Z轴待机位
LD D1302.02  ; RK_16 U6_Z 激光焊接Z轴运行条件
OUT TR0
AND H125.01  ; RK_16 U6_Z 激光焊接Z轴回原点记忆
AND D1302.14  ; RK_16 U6_Z 激光焊接Z轴手自动运行条件
ANDNOT 862.00  ; RK_16 U6_Z 激光焊接Z轴待机位标志
OUT TR1
AND W1.00  ; 手动模式
ANDNOT D1303.00  ; RK_16 焊接机构单步/自动循环运行中（总）
OUT TR2
LD 762.00  ; RK_16 U6_Z 激光焊接Z轴待机位[SW]
OR D1317.02  ; RK_16 U6_Z 激光焊接Z轴待机位（复位）
ANDLD
ANDNOT 2074.13  ; RK_16 U6_Z 激光焊接Z轴忙标志位
ANDNOT W316.14  ; RK_16 U6_Z 激光焊接Z轴轴忙标志
DIFU(013) 362.00  ; RK_16 U6_Z 激光焊接Z轴待机位[Pls]
LD TR2
LD 362.00  ; RK_16 U6_Z 激光焊接Z轴待机位[Pls]
OR 462.00  ; RK_16 U6_Z 激光焊接Z轴待机位[M]
ANDLD
ANDNOT W316.02  ; RK_16 U6_Z 激光焊接Z轴待机位完成标志
OUT 462.00  ; RK_16 U6_Z 激光焊接Z轴待机位[M]
LD TR1
LD W1.01  ; 自动模式
AND D1303.00  ; RK_16 焊接机构单步/自动循环运行中（总）
OR W319.00  ; RK_16 焊接机构单步标志
ANDLD
OUT TR2
AND D1306.05  ; RK_16 焊接机构Z轴待机位（步）
ANDNOT 2074.13  ; RK_16 U6_Z 激光焊接Z轴忙标志位
ANDNOT W316.14  ; RK_16 U6_Z 激光焊接Z轴轴忙标志
OUT 562.00  ; RK_16 U6_Z 激光焊接Z轴待机位条件
TIMHX(551) 0720 D24  ; 伺服启动延时, RK_16 U6_Z 激光焊接Z轴待机位延时[A]
LD TR2
LD 562.00  ; RK_16 U6_Z 激光焊接Z轴待机位条件
AND T0720  ; RK_16 U6_Z 激光焊接Z轴待机位延时[A]
OR 662.00  ; RK_16 U6_Z 激光焊接Z轴待机位[A]
ANDLD
ANDNOT W316.02  ; RK_16 U6_Z 激光焊接Z轴待机位完成标志
OUT 662.00  ; RK_16 U6_Z 激光焊接Z轴待机位[A]
LD TR1
LD 462.00  ; RK_16 U6_Z 激光焊接Z轴待机位[M]
OR 662.00  ; RK_16 U6_Z 激光焊接Z轴待机位[A]
ANDLD
ANDNOT 2074.13  ; RK_16 U6_Z 激光焊接Z轴忙标志位
OUT 162.00  ; RK_16 U6_Z 激光焊接Z轴待机位触发
LD TR0
LD 462.00  ; RK_16 U6_Z 激光焊接Z轴待机位[M]
OR 662.00  ; RK_16 U6_Z 激光焊接Z轴待机位[A]
AND 2074.13  ; RK_16 U6_Z 激光焊接Z轴忙标志位
AND P_1s
OR 862.00  ; RK_16 U6_Z 激光焊接Z轴待机位标志
ANDLD
OUT 962.00  ; RK_16 U6_Z 激光焊接Z轴待机位[lamp]

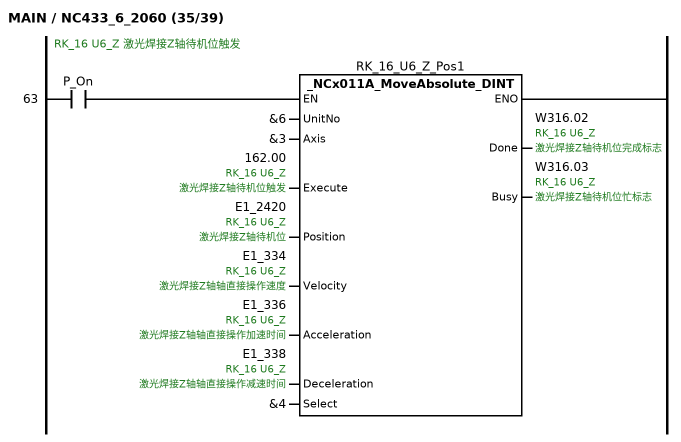
; rung 63: RK_16 U6_Z 激光焊接Z轴待机位触发
LD P_On
CALL RK_16_U6_Z_Pos1 : _NCx011A_MoveAbsolute_DINT (UnitNo := &6, Axis := &3, Execute := 162.00, Position := E1_2420, Velocity := E1_334, Acceleration := E1_336, Deceleration := E1_338, Select := &4, Done => W316.02, Busy => W316.03)  ; RK_16 U6_Z 激光焊接Z轴待机位触发, RK_16 U6_Z 激光焊接Z轴待机位, RK_16 U6_Z 激光焊接Z轴轴直接操作速度, RK_16 U6_Z 激光焊接Z轴轴直接操作加速时间, RK_16 U6_Z 激光焊接Z轴轴直接操作减速时间, RK_16 U6_Z 激光焊接Z轴待机位完成标志, RK_16 U6_Z 激光焊接Z轴待机位忙标志

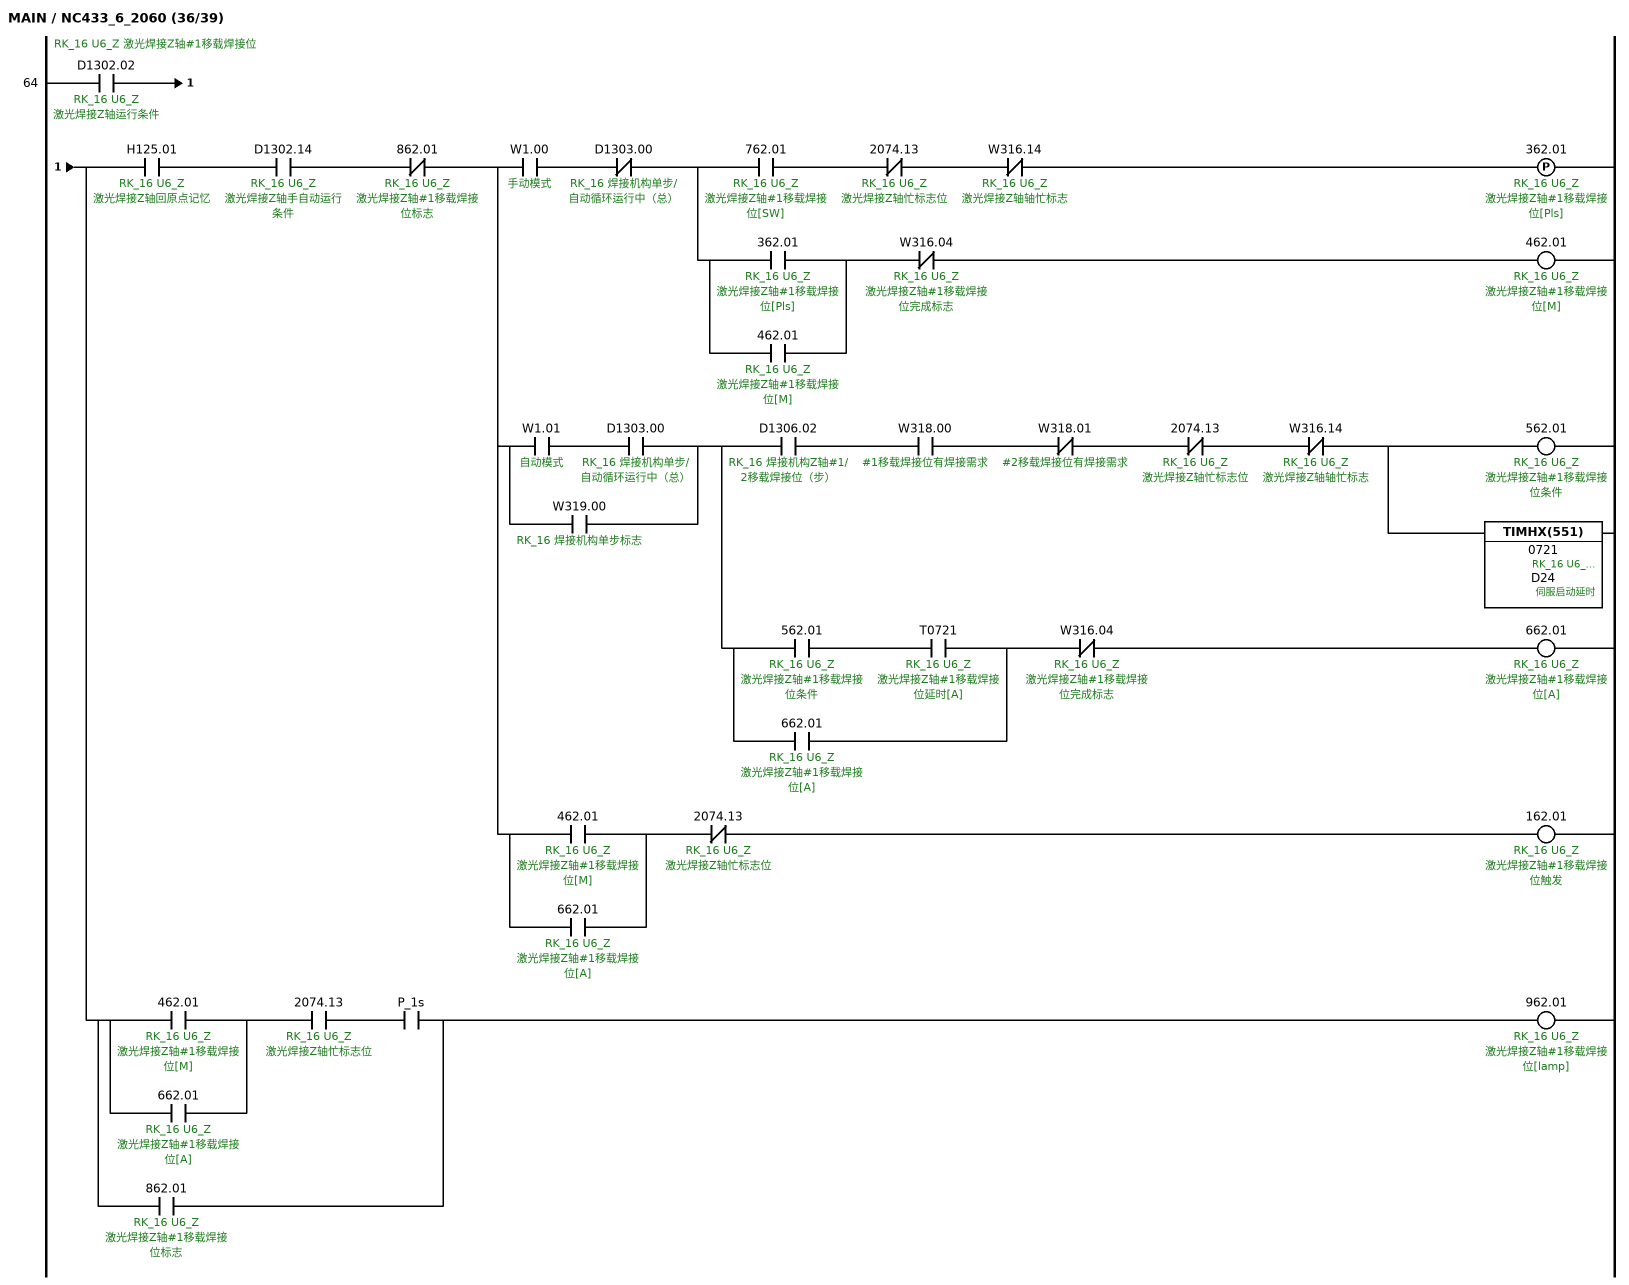
; rung 64: RK_16 U6_Z 激光焊接Z轴#1移载焊接位
LD D1302.02  ; RK_16 U6_Z 激光焊接Z轴运行条件
OUT TR0
AND H125.01  ; RK_16 U6_Z 激光焊接Z轴回原点记忆
AND D1302.14  ; RK_16 U6_Z 激光焊接Z轴手自动运行条件
ANDNOT 862.01  ; RK_16 U6_Z 激光焊接Z轴#1移载焊接位标志
OUT TR1
AND W1.00  ; 手动模式
ANDNOT D1303.00  ; RK_16 焊接机构单步/自动循环运行中（总）
OUT TR2
AND 762.01  ; RK_16 U6_Z 激光焊接Z轴#1移载焊接位[SW]
ANDNOT 2074.13  ; RK_16 U6_Z 激光焊接Z轴忙标志位
ANDNOT W316.14  ; RK_16 U6_Z 激光焊接Z轴轴忙标志
DIFU(013) 362.01  ; RK_16 U6_Z 激光焊接Z轴#1移载焊接位[Pls]
LD TR2
LD 362.01  ; RK_16 U6_Z 激光焊接Z轴#1移载焊接位[Pls]
OR 462.01  ; RK_16 U6_Z 激光焊接Z轴#1移载焊接位[M]
ANDLD
ANDNOT W316.04  ; RK_16 U6_Z 激光焊接Z轴#1移载焊接位完成标志
OUT 462.01  ; RK_16 U6_Z 激光焊接Z轴#1移载焊接位[M]
LD TR1
LD W1.01  ; 自动模式
AND D1303.00  ; RK_16 焊接机构单步/自动循环运行中（总）
OR W319.00  ; RK_16 焊接机构单步标志
ANDLD
OUT TR2
AND D1306.02  ; RK_16 焊接机构Z轴#1/2移载焊接位（步）
AND W318.00  ; #1移载焊接位有焊接需求
ANDNOT W318.01  ; #2移载焊接位有焊接需求
ANDNOT 2074.13  ; RK_16 U6_Z 激光焊接Z轴忙标志位
ANDNOT W316.14  ; RK_16 U6_Z 激光焊接Z轴轴忙标志
OUT 562.01  ; RK_16 U6_Z 激光焊接Z轴#1移载焊接位条件
TIMHX(551) 0721 D24  ; 伺服启动延时, RK_16 U6_Z 激光焊接Z轴#1移载焊接位延时[A]
LD TR2
LD 562.01  ; RK_16 U6_Z 激光焊接Z轴#1移载焊接位条件
AND T0721  ; RK_16 U6_Z 激光焊接Z轴#1移载焊接位延时[A]
OR 662.01  ; RK_16 U6_Z 激光焊接Z轴#1移载焊接位[A]
ANDLD
ANDNOT W316.04  ; RK_16 U6_Z 激光焊接Z轴#1移载焊接位完成标志
OUT 662.01  ; RK_16 U6_Z 激光焊接Z轴#1移载焊接位[A]
LD TR1
LD 462.01  ; RK_16 U6_Z 激光焊接Z轴#1移载焊接位[M]
OR 662.01  ; RK_16 U6_Z 激光焊接Z轴#1移载焊接位[A]
ANDLD
ANDNOT 2074.13  ; RK_16 U6_Z 激光焊接Z轴忙标志位
OUT 162.01  ; RK_16 U6_Z 激光焊接Z轴#1移载焊接位触发
LD TR0
LD 462.01  ; RK_16 U6_Z 激光焊接Z轴#1移载焊接位[M]
OR 662.01  ; RK_16 U6_Z 激光焊接Z轴#1移载焊接位[A]
AND 2074.13  ; RK_16 U6_Z 激光焊接Z轴忙标志位
AND P_1s
OR 862.01  ; RK_16 U6_Z 激光焊接Z轴#1移载焊接位标志
ANDLD
OUT 962.01  ; RK_16 U6_Z 激光焊接Z轴#1移载焊接位[lamp]

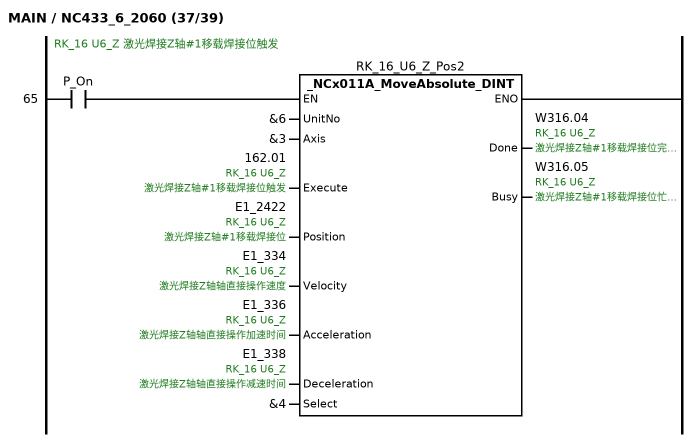
; rung 65: RK_16 U6_Z 激光焊接Z轴#1移载焊接位触发
LD P_On
CALL RK_16_U6_Z_Pos2 : _NCx011A_MoveAbsolute_DINT (UnitNo := &6, Axis := &3, Execute := 162.01, Position := E1_2422, Velocity := E1_334, Acceleration := E1_336, Deceleration := E1_338, Select := &4, Done => W316.04, Busy => W316.05)  ; RK_16 U6_Z 激光焊接Z轴#1移载焊接位触发, RK_16 U6_Z 激光焊接Z轴#1移载焊接位, RK_16 U6_Z 激光焊接Z轴轴直接操作速度, RK_16 U6_Z 激光焊接Z轴轴直接操作加速时间, RK_16 U6_Z 激光焊接Z轴轴直接操作减速时间, RK_16 U6_Z 激光焊接Z轴#1移载焊接位完成标志, RK_16 U6_Z 激光焊接Z轴#1移载焊接位忙标志

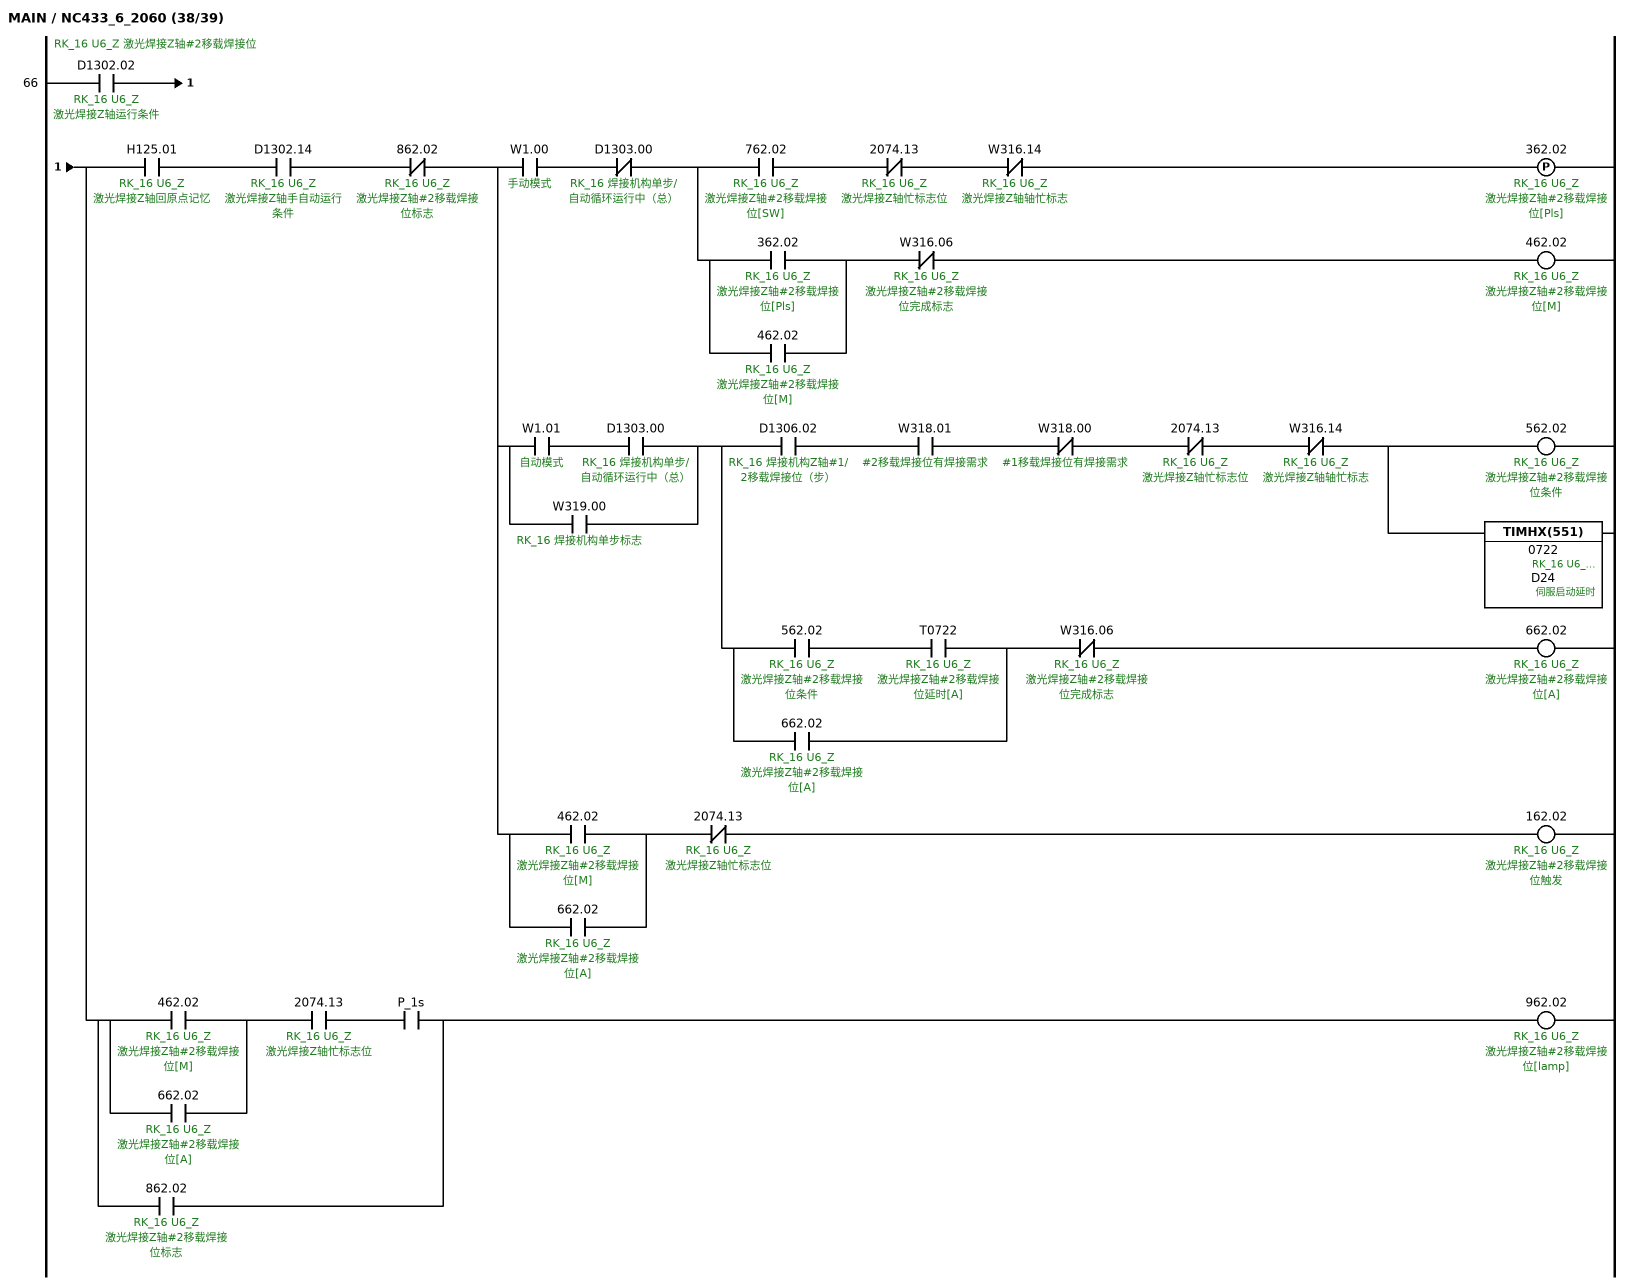
; rung 66: RK_16 U6_Z 激光焊接Z轴#2移载焊接位
LD D1302.02  ; RK_16 U6_Z 激光焊接Z轴运行条件
OUT TR0
AND H125.01  ; RK_16 U6_Z 激光焊接Z轴回原点记忆
AND D1302.14  ; RK_16 U6_Z 激光焊接Z轴手自动运行条件
ANDNOT 862.02  ; RK_16 U6_Z 激光焊接Z轴#2移载焊接位标志
OUT TR1
AND W1.00  ; 手动模式
ANDNOT D1303.00  ; RK_16 焊接机构单步/自动循环运行中（总）
OUT TR2
AND 762.02  ; RK_16 U6_Z 激光焊接Z轴#2移载焊接位[SW]
ANDNOT 2074.13  ; RK_16 U6_Z 激光焊接Z轴忙标志位
ANDNOT W316.14  ; RK_16 U6_Z 激光焊接Z轴轴忙标志
DIFU(013) 362.02  ; RK_16 U6_Z 激光焊接Z轴#2移载焊接位[Pls]
LD TR2
LD 362.02  ; RK_16 U6_Z 激光焊接Z轴#2移载焊接位[Pls]
OR 462.02  ; RK_16 U6_Z 激光焊接Z轴#2移载焊接位[M]
ANDLD
ANDNOT W316.06  ; RK_16 U6_Z 激光焊接Z轴#2移载焊接位完成标志
OUT 462.02  ; RK_16 U6_Z 激光焊接Z轴#2移载焊接位[M]
LD TR1
LD W1.01  ; 自动模式
AND D1303.00  ; RK_16 焊接机构单步/自动循环运行中（总）
OR W319.00  ; RK_16 焊接机构单步标志
ANDLD
OUT TR2
AND D1306.02  ; RK_16 焊接机构Z轴#1/2移载焊接位（步）
AND W318.01  ; #2移载焊接位有焊接需求
ANDNOT W318.00  ; #1移载焊接位有焊接需求
ANDNOT 2074.13  ; RK_16 U6_Z 激光焊接Z轴忙标志位
ANDNOT W316.14  ; RK_16 U6_Z 激光焊接Z轴轴忙标志
OUT 562.02  ; RK_16 U6_Z 激光焊接Z轴#2移载焊接位条件
TIMHX(551) 0722 D24  ; 伺服启动延时, RK_16 U6_Z 激光焊接Z轴#2移载焊接位延时[A]
LD TR2
LD 562.02  ; RK_16 U6_Z 激光焊接Z轴#2移载焊接位条件
AND T0722  ; RK_16 U6_Z 激光焊接Z轴#2移载焊接位延时[A]
OR 662.02  ; RK_16 U6_Z 激光焊接Z轴#2移载焊接位[A]
ANDLD
ANDNOT W316.06  ; RK_16 U6_Z 激光焊接Z轴#2移载焊接位完成标志
OUT 662.02  ; RK_16 U6_Z 激光焊接Z轴#2移载焊接位[A]
LD TR1
LD 462.02  ; RK_16 U6_Z 激光焊接Z轴#2移载焊接位[M]
OR 662.02  ; RK_16 U6_Z 激光焊接Z轴#2移载焊接位[A]
ANDLD
ANDNOT 2074.13  ; RK_16 U6_Z 激光焊接Z轴忙标志位
OUT 162.02  ; RK_16 U6_Z 激光焊接Z轴#2移载焊接位触发
LD TR0
LD 462.02  ; RK_16 U6_Z 激光焊接Z轴#2移载焊接位[M]
OR 662.02  ; RK_16 U6_Z 激光焊接Z轴#2移载焊接位[A]
AND 2074.13  ; RK_16 U6_Z 激光焊接Z轴忙标志位
AND P_1s
OR 862.02  ; RK_16 U6_Z 激光焊接Z轴#2移载焊接位标志
ANDLD
OUT 962.02  ; RK_16 U6_Z 激光焊接Z轴#2移载焊接位[lamp]

